LIN {X 0,Y 715.603,Z 787.704,A -85,B 0,C 180,E1 31621.98,E2 31621.98} C_VEL
LIN {X 0,Y 714.708,Z 772.954,A -85,B 0,C 180,E1 31621.864,E2 31621.864} C_VEL
LIN {X 0,Y 714.613,Z 761.128,A -85,B 0,C 180,E1 31621.852,E2 31621.852} C_VEL
LIN {X 0,Y 712.527,Z 773.661,A -85,B 0,C 180,E1 31621.581,E2 31621.581} C_VEL
LIN {X 0,Y 711.718,Z 777.536,A -85,B 0,C 180,E1 31621.475,E2 31621.475} C_VEL
LIN {X 0,Y 707.438,Z 835.712,A -85,B 0,C 180,E1 31620.904,E2 31620.904} C_VEL
LIN {X 0,Y 703.742,Z 875.337,A -85,B 0,C 180,E1 31620.398,E2 31620.398} C_VEL
LIN {X 0,Y 701.35,Z 893.858,A -85,B 0,C 180,E1 31620.063,E2 31620.063} C_VEL
LIN {X 0,Y 699.884,Z 900.884,A -85,B 0,C 180,E1 31619.855,E2 31619.855} C_VEL
LIN {X 0,Y 698.183,Z 921.476,A -85,B 0,C 180,E1 31619.675,E2 31619.675} C_VEL
LIN {X 0,Y 695.199,Z 934.998,A -85,B 0,C 180,E1 31619.546,E2 31619.546} C_VEL
LIN {X 0,Y 691.805,Z 945.388,A -85,B 0,C 180,E1 31619.339,E2 31619.339} C_VEL
LIN {X 0,Y 689.317,Z 952.203,A -85,B 0,C 180,E1 31619.075,E2 31619.075} C_VEL
LIN {X 0,Y 688.817,Z 954.108,A -85,B 0,C 180,E1 31618.988,E2 31618.988} C_VEL
LIN {X 0,Y 688.302,Z 1018.799,A -85,B 0,C 180,E1 31618.229,E2 31618.229} C_VEL
LIN {X 0,Y 687.827,Z 1042.443,A -85,B 0,C 180,E1 31617.796,E2 31617.796} C_VEL
LIN {X 0,Y 687.249,Z 1065.699,A -85,B 0,C 180,E1 31617.208,E2 31617.208} C_VEL
LIN {X 0,Y 686.594,Z 1087.292,A -85,B 0,C 180,E1 31616.511,E2 31616.511} C_VEL
LIN {X 0,Y 685.818,Z 1109.823,A -85,B 0,C 180,E1 31615.613,E2 31615.613} C_VEL
LIN {X 0,Y 685.018,Z 1130.719,A -85,B 0,C 180,E1 31614.616,E2 31614.616} C_VEL
LIN {X 0,Y 684.173,Z 1151.786,A -85,B 0,C 180,E1 31613.424,E2 31613.424} C_VEL
LIN {X 0,Y 683.335,Z 1171.979,A -85,B 0,C 180,E1 31612.09,E2 31612.09} C_VEL
LIN {X 0,Y 682.504,Z 1192.49,A -85,B 0,C 180,E1 31610.497,E2 31610.497} C_VEL
LIN {X 0,Y 681.903,Z 1208.158,A -85,B 0,C 180,E1 31609.087,E2 31609.087} C_VEL
LIN {X 0,Y 681.353,Z 1223.561,A -85,B 0,C 180,E1 31607.509,E2 31607.509} C_VEL
LIN {X 0,Y 680.853,Z 1238.91,A -85,B 0,C 180,E1 31605.678,E2 31605.678} C_VEL
LIN {X 0,Y 680.524,Z 1251.279,A -85,B 0,C 180,E1 31603.944,E2 31603.944} C_VEL
LIN {X 0,Y 680.275,Z 1262.038,A -85,B 0,C 180,E1 31602.192,E2 31602.192} C_VEL
LIN {X 0,Y 680.096,Z 1271.99,A -85,B 0,C 180,E1 31600.248,E2 31600.248} C_VEL
LIN {X 0,Y 679.995,Z 1280.024,A -85,B 0,C 180,E1 31598.286,E2 31598.286} C_VEL
LIN {X 0,Y 679.928,Z 1285.324,A -85,B 0,C 180,E1 31596.673,E2 31596.673} C_VEL
LIN {X 0,Y 679.901,Z 1290.199,A -85,B 0,C 180,E1 31594.725,E2 31594.725} C_VEL
LIN {X 0,Y 679.894,Z 1293.515,A -85,B 0,C 180,E1 31592.614,E2 31592.614} C_VEL
LIN {X 0,Y 679.899,Z 1294.802,A -85,B 0,C 180,E1 31590.76,E2 31590.76} C_VEL
LIN {X 0,Y 679.909,Z 1294.747,A -85,B 0,C 180,E1 31589.074,E2 31589.074} C_VEL
LIN {X 0,Y 679.908,Z 1293.103,A -85,B 0,C 180,E1 31587.051,E2 31587.051} C_VEL
LIN {X 0,Y 679.914,Z 1289.645,A -85,B 0,C 180,E1 31585.024,E2 31585.024} C_VEL
LIN {X 0,Y 679.926,Z 1285.068,A -85,B 0,C 180,E1 31583.245,E2 31583.245} C_VEL
LIN {X 0,Y 679.998,Z 1279.731,A -85,B 0,C 180,E1 31581.631,E2 31581.631} C_VEL
LIN {X 0,Y 680.106,Z 1271.598,A -85,B 0,C 180,E1 31579.669,E2 31579.669} C_VEL
LIN {X 0,Y 680.285,Z 1261.402,A -85,B 0,C 180,E1 31577.696,E2 31577.696} C_VEL
LIN {X 0,Y 680.523,Z 1251.281,A -85,B 0,C 180,E1 31576.058,E2 31576.058} C_VEL
LIN {X 0,Y 680.808,Z 1240.215,A -85,B 0,C 180,E1 31574.498,E2 31574.498} C_VEL
LIN {X 0,Y 681.277,Z 1225.94,A -85,B 0,C 180,E1 31572.756,E2 31572.756} C_VEL
LIN {X 0,Y 681.837,Z 1210.008,A -85,B 0,C 180,E1 31571.091,E2 31571.091} C_VEL
LIN {X 0,Y 682.375,Z 1195.578,A -85,B 0,C 180,E1 31569.77,E2 31569.77} C_VEL
LIN {X 0,Y 683.11,Z 1178.049,A -85,B 0,C 180,E1 31568.353,E2 31568.353} C_VEL
LIN {X 0,Y 683.906,Z 1158.295,A -85,B 0,C 180,E1 31566.979,E2 31566.979} C_VEL
LIN {X 0,Y 684.734,Z 1138.058,A -85,B 0,C 180,E1 31565.776,E2 31565.776} C_VEL
LIN {X 0,Y 685.55,Z 1116.849,A -85,B 0,C 180,E1 31564.702,E2 31564.702} C_VEL
LIN {X 0,Y 686.328,Z 1095.82,A -85,B 0,C 180,E1 31563.806,E2 31563.806} C_VEL
LIN {X 0,Y 687.009,Z 1073.239,A -85,B 0,C 180,E1 31563.019,E2 31563.019} C_VEL
LIN {X 0,Y 687.673,Z 1050.257,A -85,B 0,C 180,E1 31562.385,E2 31562.385} C_VEL
LIN {X 0,Y 688.127,Z 1026.734,A -85,B 0,C 180,E1 31561.899,E2 31561.899} C_VEL
LIN {X 0,Y 688.49,Z 1000.263,A -85,B 0,C 180,E1 31561.535,E2 31561.535} C_VEL
LIN {X 0,Y 688.848,Z 953.484,A -85,B 0,C 180,E1 31561.001,E2 31561.001} C_VEL
LIN {X 0,Y 691.067,Z 947.432,A -85,B 0,C 180,E1 31560.724,E2 31560.724} C_VEL
LIN {X 0,Y 694.4,Z 937.673,A -85,B 0,C 180,E1 31560.494,E2 31560.494} C_VEL
LIN {X 0,Y 697.652,Z 924.638,A -85,B 0,C 180,E1 31560.35,E2 31560.35} C_VEL
LIN {X 0,Y 699.303,Z 910.098,A -85,B 0,C 180,E1 31560.228,E2 31560.228} C_VEL
LIN {X 0,Y 700.088,Z 899.542,A -85,B 0,C 180,E1 31560.116,E2 31560.116} C_VEL
LIN {X 0,Y 701.619,Z 892.218,A -85,B 0,C 180,E1 31559.899,E2 31559.899} C_VEL
LIN {X 0,Y 704.219,Z 870.835,A -85,B 0,C 180,E1 31559.536,E2 31559.536} C_VEL
LIN {X 0,Y 708.05,Z 828.181,A -85,B 0,C 180,E1 31559.013,E2 31559.013} C_VEL
LIN {X 0,Y 711.957,Z 775.957,A -85,B 0,C 180,E1 31558.494,E2 31558.494} C_VEL
LIN {X 0,Y 713.841,Z 766.512,A -85,B 0,C 180,E1 31558.248,E2 31558.248} C_VEL
LIN {X 0,Y 714.629,Z 761.008,A -85,B 0,C 180,E1 31558.146,E2 31558.146} C_VEL
LIN {X 0,Y 714.92,Z 778.455,A -85,B 0,C 180,E1 31558.108,E2 31558.108} C_VEL
LIN {X 0,Y 716.169,Z 792.802,A -85,B 0,C 180,E1 31557.948,E2 31557.948} C_VEL
LIN {X 0,Y 718.366,Z 806.064,A -85,B 0,C 180,E1 31557.669,E2 31557.669} C_VEL
LIN {X 0,Y 721.525,Z 818.398,A -85,B 0,C 180,E1 31557.275,E2 31557.275} C_VEL
LIN {X 0,Y 725.606,Z 829.571,A -85,B 0,C 180,E1 31556.777,E2 31556.777} C_VEL
LIN {X 0,Y 730.214,Z 839.109,A -85,B 0,C 180,E1 31556.203,E2 31556.203} C_VEL
LIN {X 0,Y 731.525,Z 843.469,A -85,B 0,C 180,E1 31555.81,E2 31555.81} C_VEL
LIN {X 0,Y 731.39,Z 846.84,A -85,B 0,C 180,E1 31555.387,E2 31555.387} C_VEL
LIN {X 0,Y 730.13,Z 849.08,A -85,B 0,C 180,E1 31554.979,E2 31554.979} C_VEL
LIN {X 0,Y 727.783,Z 850.434,A -85,B 0,C 180,E1 31554.559,E2 31554.559} C_VEL
LIN {X 0,Y 724.29,Z 850.661,A -85,B 0,C 180,E1 31554.132,E2 31554.132} C_VEL
LIN {X 0,Y 720.235,Z 849.65,A -85,B 0,C 180,E1 31553.765,E2 31553.765} C_VEL
LIN {X 0,Y 711.761,Z 845.351,A -85,B 0,C 180,E1 31553.067,E2 31553.067} C_VEL
LIN {X 0,Y 704.753,Z 839.928,A -85,B 0,C 180,E1 31552.343,E2 31552.343} C_VEL
LIN {X 0,Y 698.647,Z 832.828,A -85,B 0,C 180,E1 31551.523,E2 31551.523} C_VEL
LIN {X 0,Y 694.056,Z 824.409,A -85,B 0,C 180,E1 31550.665,E2 31550.665} C_VEL
LIN {X 0,Y 690.733,Z 814.145,A -85,B 0,C 180,E1 31549.719,E2 31549.719} C_VEL
LIN {X 0,Y 689.006,Z 801.685,A -85,B 0,C 180,E1 31548.68,E2 31548.68} C_VEL
LIN {X 0,Y 688.911,Z 784.149,A -85,B 0,C 180,E1 31547.33,E2 31547.33} C_VEL
LIN {X 0,Y 690.246,Z 746.13,A -85,B 0,C 180,E1 31544.428,E2 31544.428} C_VEL
LIN {X 0,Y 691.594,Z 709.846,A -85,B 0,C 180,E1 31541.576,E2 31541.576} C_VEL
LIN {X 0,Y 692.854,Z 674.643,A -85,B 0,C 180,E1 31538.727,E2 31538.727} C_VEL
LIN {X 0,Y 694.016,Z 640.169,A -85,B 0,C 180,E1 31535.845,E2 31535.845} C_VEL
LIN {X 0,Y 694.079,Z 634.852,A -85,B 0,C 180,E1 31535.378,E2 31535.378} C_VEL
LIN {X 0,Y 685.307,Z 614.541,A -85,B 0,C 180,E1 31532.773,E2 31532.773} C_VEL
LIN {X 0,Y 681.315,Z 605.83,A -85,B 0,C 180,E1 31531.596,E2 31531.596} C_VEL
LIN {X 0,Y 680.505,Z 603.217,A -85,B 0,C 180,E1 31531.244,E2 31531.244} C_VEL
LIN {X 0,Y 680.512,Z 603.214,A -85,B 0,C 180,E1 31528.333,E2 31528.333} C_VEL
LIN {X 0,Y 680.516,Z 603.213,A -85,B 0,C 180,E1 31525.314,E2 31525.314} C_VEL
LIN {X 0,Y 680.519,Z 603.213,A -85,B 0,C 180,E1 31522.237,E2 31522.237} C_VEL
LIN {X 0,Y 680.52,Z 603.21,A -85,B 0,C 180,E1 31519.127,E2 31519.127} C_VEL
LIN {X 0,Y 680.521,Z 603.213,A -85,B 0,C 180,E1 31516.035,E2 31516.035} C_VEL
LIN {X 0,Y 680.524,Z 603.212,A -85,B 0,C 180,E1 31512.991,E2 31512.991} C_VEL
LIN {X 0,Y 680.526,Z 603.215,A -85,B 0,C 180,E1 31509.899,E2 31509.899} C_VEL
LIN {X 0,Y 680.53,Z 603.213,A -85,B 0,C 180,E1 31506.835,E2 31506.835} C_VEL
LIN {X 0,Y 680.515,Z 603.214,A -85,B 0,C 180,E1 31503.791,E2 31503.791} C_VEL
LIN {X 0,Y 680.511,Z 603.212,A -85,B 0,C 180,E1 31500.758,E2 31500.758} C_VEL
LIN {X 0,Y 680.505,Z 603.211,A -85,B 0,C 180,E1 31497.811,E2 31497.811} C_VEL
LIN {X 0,Y 680.504,Z 603.211,A -85,B 0,C 180,E1 31494.858,E2 31494.858} C_VEL
LIN {X 0,Y 680.508,Z 603.211,A -85,B 0,C 180,E1 31491.891,E2 31491.891} C_VEL
LIN {X 0,Y 680.515,Z 603.211,A -85,B 0,C 180,E1 31488.902,E2 31488.902} C_VEL
LIN {X 0,Y 680.522,Z 603.212,A -85,B 0,C 180,E1 31485.86,E2 31485.86} C_VEL
LIN {X 0,Y 680.521,Z 603.213,A -85,B 0,C 180,E1 31482.734,E2 31482.734} C_VEL
LIN {X 0,Y 680.524,Z 603.213,A -85,B 0,C 180,E1 31479.711,E2 31479.711} C_VEL
LIN {X 0,Y 680.526,Z 603.212,A -85,B 0,C 180,E1 31476.627,E2 31476.627} C_VEL
LIN {X 0,Y 680.522,Z 603.215,A -85,B 0,C 180,E1 31473.564,E2 31473.564} C_VEL
LIN {X 0,Y 680.511,Z 603.214,A -85,B 0,C 180,E1 31470.607,E2 31470.607} C_VEL
LIN {X 0,Y 680.52,Z 603.208,A -85,B 0,C 180,E1 31469.429,E2 31469.429} C_VEL
LIN {X 0,Y 679.55,Z 603.333,A -85,B 0,C 180,E1 31468.78,E2 31468.78} C_VEL
LIN {X 0,Y 673.093,Z 604.139,A -85,B 0,C 180,E1 31466.963,E2 31466.963} C_VEL
LIN {X 0,Y 672.574,Z 604.199,A -85,B 0,C 180,E1 31466.49,E2 31466.49} C_VEL
LIN {X 0,Y 672.566,Z 604.202,A -85,B 0,C 180,E1 31463.511,E2 31463.511} C_VEL
LIN {X 0,Y 672.583,Z 604.204,A -85,B 0,C 180,E1 31460.595,E2 31460.595} C_VEL
LIN {X 0,Y 672.576,Z 604.194,A -85,B 0,C 180,E1 31457.55,E2 31457.55} C_VEL
LIN {X 0,Y 672.586,Z 604.2,A -85,B 0,C 180,E1 31454.56,E2 31454.56} C_VEL
LIN {X 0,Y 672.591,Z 604.193,A -85,B 0,C 180,E1 31451.416,E2 31451.416} C_VEL
LIN {X 0,Y 672.579,Z 604.203,A -85,B 0,C 180,E1 31448.283,E2 31448.283} C_VEL
LIN {X 0,Y 672.591,Z 604.204,A -85,B 0,C 180,E1 31445.15,E2 31445.15} C_VEL
LIN {X 0,Y 672.576,Z 604.205,A -85,B 0,C 180,E1 31442.053,E2 31442.053} C_VEL
LIN {X 0,Y 672.594,Z 604.397,A -85,B 0,C 180,E1 31440.786,E2 31440.786} C_VEL
LIN {X 0,Y 677.704,Z 621.502,A -85,B 0,C 180,E1 31439.484,E2 31439.484} C_VEL
LIN {X 0,Y 677.378,Z 660.167,A -85,B 0,C 180,E1 31436.945,E2 31436.945} C_VEL
LIN {X 0,Y 676.584,Z 704.691,A -85,B 0,C 180,E1 31433.978,E2 31433.978} C_VEL
LIN {X 0,Y 675.775,Z 749.981,A -85,B 0,C 180,E1 31430.98,E2 31430.98} C_VEL
LIN {X 0,Y 674.803,Z 795.336,A -85,B 0,C 180,E1 31427.95,E2 31427.95} C_VEL
LIN {X 0,Y 674.169,Z 831.281,A -85,B 0,C 180,E1 31425.589,E2 31425.589} C_VEL
LIN {X 0,Y 675.101,Z 841.648,A -85,B 0,C 180,E1 31425.451,E2 31425.451} C_VEL
LIN {X 0,Y 674.416,Z 1000.774,A -85,B 0,C 180,E1 31423.715,E2 31423.715} C_VEL
LIN {X 0,Y 674.227,Z 1018.235,A -85,B 0,C 180,E1 31423.37,E2 31423.37} C_VEL
LIN {X 0,Y 673.939,Z 1035.447,A -85,B 0,C 180,E1 31422.857,E2 31422.857} C_VEL
LIN {X 0,Y 673.617,Z 1051.632,A -85,B 0,C 180,E1 31422.21,E2 31422.21} C_VEL
LIN {X 0,Y 673.284,Z 1066.92,A -85,B 0,C 180,E1 31421.43,E2 31421.43} C_VEL
LIN {X 0,Y 672.954,Z 1081.016,A -85,B 0,C 180,E1 31420.529,E2 31420.529} C_VEL
LIN {X 0,Y 672.636,Z 1094.67,A -85,B 0,C 180,E1 31419.453,E2 31419.453} C_VEL
LIN {X 0,Y 672.382,Z 1106.683,A -85,B 0,C 180,E1 31418.292,E2 31418.292} C_VEL
LIN {X 0,Y 672.193,Z 1116.775,A -85,B 0,C 180,E1 31417.091,E2 31417.091} C_VEL
LIN {X 0,Y 672.051,Z 1125.967,A -85,B 0,C 180,E1 31415.72,E2 31415.72} C_VEL
LIN {X 0,Y 671.974,Z 1133.125,A -85,B 0,C 180,E1 31414.351,E2 31414.351} C_VEL
LIN {X 0,Y 671.934,Z 1138.766,A -85,B 0,C 180,E1 31412.899,E2 31412.899} C_VEL
LIN {X 0,Y 671.917,Z 1142.505,A -85,B 0,C 180,E1 31411.448,E2 31411.448} C_VEL
LIN {X 0,Y 671.924,Z 1144.6,A -85,B 0,C 180,E1 31409.914,E2 31409.914} C_VEL
LIN {X 0,Y 671.914,Z 1144.855,A -85,B 0,C 180,E1 31408.379,E2 31408.379} C_VEL
LIN {X 0,Y 671.919,Z 1143.303,A -85,B 0,C 180,E1 31406.892,E2 31406.892} C_VEL
LIN {X 0,Y 671.925,Z 1139.885,A -85,B 0,C 180,E1 31405.39,E2 31405.39} C_VEL
LIN {X 0,Y 671.96,Z 1134.758,A -85,B 0,C 180,E1 31403.934,E2 31403.934} C_VEL
LIN {X 0,Y 672.026,Z 1128.128,A -85,B 0,C 180,E1 31402.561,E2 31402.561} C_VEL
LIN {X 0,Y 672.14,Z 1120.07,A -85,B 0,C 180,E1 31401.271,E2 31401.271} C_VEL
LIN {X 0,Y 672.316,Z 1109.903,A -85,B 0,C 180,E1 31399.978,E2 31399.978} C_VEL
LIN {X 0,Y 672.56,Z 1098.153,A -85,B 0,C 180,E1 31398.768,E2 31398.768} C_VEL
LIN {X 0,Y 672.86,Z 1085.21,A -85,B 0,C 180,E1 31397.686,E2 31397.686} C_VEL
LIN {X 0,Y 673.185,Z 1071.123,A -85,B 0,C 180,E1 31396.733,E2 31396.733} C_VEL
LIN {X 0,Y 673.522,Z 1056.055,A -85,B 0,C 180,E1 31395.908,E2 31395.908} C_VEL
LIN {X 0,Y 673.857,Z 1039.951,A -85,B 0,C 180,E1 31395.212,E2 31395.212} C_VEL
LIN {X 0,Y 674.151,Z 1022.973,A -85,B 0,C 180,E1 31394.666,E2 31394.666} C_VEL
LIN {X 0,Y 674.374,Z 1004.976,A -85,B 0,C 180,E1 31394.264,E2 31394.264} C_VEL
LIN {X 0,Y 674.515,Z 984.639,A -85,B 0,C 180,E1 31393.999,E2 31393.999} C_VEL
LIN {X 0,Y 674.892,Z 837.233,A -85,B 0,C 180,E1 31392.406,E2 31392.406} C_VEL
LIN {X 0,Y 674.157,Z 830.801,A -85,B 0,C 180,E1 31392.298,E2 31392.298} C_VEL
LIN {X 0,Y 675.054,Z 785.156,A -85,B 0,C 180,E1 31389.267,E2 31389.267} C_VEL
LIN {X 0,Y 675.759,Z 751.14,A -85,B 0,C 180,E1 31387.005,E2 31387.005} C_VEL
LIN {X 0,Y 676.57,Z 705.123,A -85,B 0,C 180,E1 31383.963,E2 31383.963} C_VEL
LIN {X 0,Y 677.378,Z 659.877,A -85,B 0,C 180,E1 31380.945,E2 31380.945} C_VEL
LIN {X 0,Y 677.729,Z 621.412,A -85,B 0,C 180,E1 31378.415,E2 31378.415} C_VEL
LIN {X 0,Y 672.578,Z 604.201,A -85,B 0,C 180,E1 31377.086,E2 31377.086} C_VEL
LIN {X 0,Y 672.567,Z 604.197,A -85,B 0,C 180,E1 31374.038,E2 31374.038} C_VEL
LIN {X 0,Y 672.588,Z 604.195,A -85,B 0,C 180,E1 31371.033,E2 31371.033} C_VEL
LIN {X 0,Y 672.567,Z 604.198,A -85,B 0,C 180,E1 31368.009,E2 31368.009} C_VEL
LIN {X 0,Y 672.576,Z 604.202,A -85,B 0,C 180,E1 31365.044,E2 31365.044} C_VEL
LIN {X 0,Y 672.584,Z 604.196,A -85,B 0,C 180,E1 31361.984,E2 31361.984} C_VEL
LIN {X 0,Y 672.579,Z 604.2,A -85,B 0,C 180,E1 31358.856,E2 31358.856} C_VEL
LIN {X 0,Y 672.589,Z 604.203,A -85,B 0,C 180,E1 31355.75,E2 31355.75} C_VEL
LIN {X 0,Y 672.583,Z 604.204,A -85,B 0,C 180,E1 31352.66,E2 31352.66} C_VEL
LIN {X 0,Y 672.579,Z 604.3,A -85,B 0,C 180,E1 31350.233,E2 31350.233} C_VEL
LIN {X 0,Y 672.874,Z 605.616,A -85,B 0,C 180,E1 31350.149,E2 31350.149} C_VEL
LIN {X 0,Y 674.8,Z 608.814,A -85,B 0,C 180,E1 31349.992,E2 31349.992} C_VEL
LIN {X 0,Y 683.922,Z 625.294,A -85,B 0,C 180,E1 31349.274,E2 31349.274} C_VEL
LIN {X 0,Y 681.83,Z 883.098,A -85,B 0,C 180,E1 31346.28,E2 31346.28} C_VEL
LIN {X 0,Y 681.257,Z 946.678,A -85,B 0,C 180,E1 31345.528,E2 31345.528} C_VEL
LIN {X 0,Y 680.809,Z 970.073,A -85,B 0,C 180,E1 31345.119,E2 31345.119} C_VEL
LIN {X 0,Y 680.146,Z 992.867,A -85,B 0,C 180,E1 31344.552,E2 31344.552} C_VEL
LIN {X 0,Y 679.55,Z 1011.718,A -85,B 0,C 180,E1 31343.961,E2 31343.961} C_VEL
LIN {X 0,Y 678.871,Z 1029.536,A -85,B 0,C 180,E1 31343.295,E2 31343.295} C_VEL
LIN {X 0,Y 678.195,Z 1046.859,A -85,B 0,C 180,E1 31342.54,E2 31342.54} C_VEL
LIN {X 0,Y 677.316,Z 1067.83,A -85,B 0,C 180,E1 31341.476,E2 31341.476} C_VEL
LIN {X 0,Y 676.37,Z 1088.323,A -85,B 0,C 180,E1 31340.239,E2 31340.239} C_VEL
LIN {X 0,Y 675.609,Z 1104.819,A -85,B 0,C 180,E1 31339.092,E2 31339.092} C_VEL
LIN {X 0,Y 674.944,Z 1119.984,A -85,B 0,C 180,E1 31337.903,E2 31337.903} C_VEL
LIN {X 0,Y 674.231,Z 1136.28,A -85,B 0,C 180,E1 31336.455,E2 31336.455} C_VEL
LIN {X 0,Y 673.511,Z 1154.036,A -85,B 0,C 180,E1 31334.619,E2 31334.619} C_VEL
LIN {X 0,Y 673.049,Z 1167.097,A -85,B 0,C 180,E1 31333.051,E2 31333.051} C_VEL
LIN {X 0,Y 672.652,Z 1179.65,A -85,B 0,C 180,E1 31331.316,E2 31331.316} C_VEL
LIN {X 0,Y 672.338,Z 1191.404,A -85,B 0,C 180,E1 31329.415,E2 31329.415} C_VEL
LIN {X 0,Y 672.128,Z 1201.454,A -85,B 0,C 180,E1 31327.436,E2 31327.436} C_VEL
LIN {X 0,Y 672.003,Z 1209.282,A -85,B 0,C 180,E1 31325.55,E2 31325.55} C_VEL
LIN {X 0,Y 671.948,Z 1215.203,A -85,B 0,C 180,E1 31323.754,E2 31323.754} C_VEL
LIN {X 0,Y 671.916,Z 1220.399,A -85,B 0,C 180,E1 31321.62,E2 31321.62} C_VEL
LIN {X 0,Y 671.904,Z 1223.334,A -85,B 0,C 180,E1 31319.744,E2 31319.744} C_VEL
LIN {X 0,Y 671.904,Z 1224.787,A -85,B 0,C 180,E1 31317.783,E2 31317.783} C_VEL
LIN {X 0,Y 671.912,Z 1224.731,A -85,B 0,C 180,E1 31315.989,E2 31315.989} C_VEL
LIN {X 0,Y 671.919,Z 1223.059,A -85,B 0,C 180,E1 31313.935,E2 31313.935} C_VEL
LIN {X 0,Y 671.928,Z 1219.534,A -85,B 0,C 180,E1 31311.873,E2 31311.873} C_VEL
LIN {X 0,Y 671.955,Z 1214.979,A -85,B 0,C 180,E1 31310.091,E2 31310.091} C_VEL
LIN {X 0,Y 672.005,Z 1209.462,A -85,B 0,C 180,E1 31308.412,E2 31308.412} C_VEL
LIN {X 0,Y 672.128,Z 1201.571,A -85,B 0,C 180,E1 31306.493,E2 31306.493} C_VEL
LIN {X 0,Y 672.337,Z 1191.242,A -85,B 0,C 180,E1 31304.473,E2 31304.473} C_VEL
LIN {X 0,Y 672.608,Z 1180.95,A -85,B 0,C 180,E1 31302.793,E2 31302.793} C_VEL
LIN {X 0,Y 672.957,Z 1169.634,A -85,B 0,C 180,E1 31301.19,E2 31301.19} C_VEL
LIN {X 0,Y 673.434,Z 1156.207,A -85,B 0,C 180,E1 31299.536,E2 31299.536} C_VEL
LIN {X 0,Y 674.137,Z 1138.647,A -85,B 0,C 180,E1 31297.685,E2 31297.685} C_VEL
LIN {X 0,Y 674.778,Z 1123.633,A -85,B 0,C 180,E1 31296.314,E2 31296.314} C_VEL
LIN {X 0,Y 675.517,Z 1107.29,A -85,B 0,C 180,E1 31295.001,E2 31295.001} C_VEL
LIN {X 0,Y 676.327,Z 1089.423,A -85,B 0,C 180,E1 31293.741,E2 31293.741} C_VEL
LIN {X 0,Y 677.304,Z 1067.704,A -85,B 0,C 180,E1 31292.431,E2 31292.431} C_VEL
LIN {X 0,Y 678.102,Z 1048.803,A -85,B 0,C 180,E1 31291.461,E2 31291.461} C_VEL
LIN {X 0,Y 678.798,Z 1031.547,A -85,B 0,C 180,E1 31290.697,E2 31290.697} C_VEL
LIN {X 0,Y 679.463,Z 1013.908,A -85,B 0,C 180,E1 31290.026,E2 31290.026} C_VEL
LIN {X 0,Y 680.056,Z 995.914,A -85,B 0,C 180,E1 31289.448,E2 31289.448} C_VEL
LIN {X 0,Y 680.649,Z 975.131,A -85,B 0,C 180,E1 31288.906,E2 31288.906} C_VEL
LIN {X 0,Y 681.229,Z 949.547,A -85,B 0,C 180,E1 31288.422,E2 31288.422} C_VEL
LIN {X 0,Y 681.625,Z 909.928,A -85,B 0,C 180,E1 31287.937,E2 31287.937} C_VEL
LIN {X 0,Y 683.667,Z 645.309,A -85,B 0,C 180,E1 31284.885,E2 31284.885} C_VEL
LIN {X 0,Y 683.579,Z 624.804,A -85,B 0,C 180,E1 31284.653,E2 31284.653} C_VEL
LIN {X 0,Y 675.913,Z 612.154,A -85,B 0,C 180,E1 31284.244,E2 31284.244} C_VEL
LIN {X 0,Y 675.178,Z 610.975,A -85,B 0,C 180,E1 31283.386,E2 31283.386} C_VEL
LIN {X 0,Y 675.379,Z 611.387,A -85,B 0,C 180,E1 31282.199,E2 31282.199} C_VEL
LIN {X 0,Y 676.034,Z 612.93,A -85,B 0,C 180,E1 31281.271,E2 31281.271} C_VEL
LIN {X 0,Y 677.44,Z 616.483,A -85,B 0,C 180,E1 31280.055,E2 31280.055} C_VEL
LIN {X 0,Y 678.902,Z 620.462,A -85,B 0,C 180,E1 31279.161,E2 31279.161} C_VEL
LIN {X 0,Y 679.568,Z 622.879,A -85,B 0,C 180,E1 31278.753,E2 31278.753} C_VEL
LIN {X 0,Y 676.672,Z 634.327,A -85,B 0,C 180,E1 31277.752,E2 31277.752} C_VEL
LIN {X 0,Y 674.724,Z 648.114,A -85,B 0,C 180,E1 31276.756,E2 31276.756} C_VEL
LIN {X 0,Y 673.436,Z 666.247,A -85,B 0,C 180,E1 31275.66,E2 31275.66} C_VEL
LIN {X 0,Y 672.583,Z 694.895,A -85,B 0,C 180,E1 31274.161,E2 31274.161} C_VEL
LIN {X 0,Y 672.595,Z 770.126,A -85,B 0,C 180,E1 31270.516,E2 31270.516} C_VEL
LIN {X 0,Y 674.512,Z 789.281,A -85,B 0,C 180,E1 31269.57,E2 31269.57} C_VEL
LIN {X 0,Y 677.902,Z 804.887,A -85,B 0,C 180,E1 31268.782,E2 31268.782} C_VEL
LIN {X 0,Y 682.915,Z 818.369,A -85,B 0,C 180,E1 31268.095,E2 31268.095} C_VEL
LIN {X 0,Y 689.341,Z 830.207,A -85,B 0,C 180,E1 31267.493,E2 31267.493} C_VEL
LIN {X 0,Y 697.093,Z 840.45,A -85,B 0,C 180,E1 31266.97,E2 31266.97} C_VEL
LIN {X 0,Y 705.641,Z 848.966,A -85,B 0,C 180,E1 31266.54,E2 31266.54} C_VEL
LIN {X 0,Y 710.972,Z 853.164,A -85,B 0,C 180,E1 31266.307,E2 31266.307} C_VEL
LIN {X 0,Y 715.788,Z 855.733,A -85,B 0,C 180,E1 31266.02,E2 31266.02} C_VEL
LIN {X 0,Y 720.755,Z 857.13,A -85,B 0,C 180,E1 31265.615,E2 31265.615} C_VEL
LIN {X 0,Y 724.417,Z 857.036,A -85,B 0,C 180,E1 31265.202,E2 31265.202} C_VEL
LIN {X 0,Y 726.939,Z 855.868,A -85,B 0,C 180,E1 31264.798,E2 31264.798} C_VEL
LIN {X 0,Y 728.59,Z 853.457,A -85,B 0,C 180,E1 31264.336,E2 31264.336} C_VEL
LIN {X 0,Y 728.825,Z 849.868,A -85,B 0,C 180,E1 31263.877,E2 31263.877} C_VEL
LIN {X 0,Y 727.476,Z 845.421,A -85,B 0,C 180,E1 31263.471,E2 31263.471} C_VEL
LIN {X 0,Y 722.555,Z 835.393,A -85,B 0,C 180,E1 31262.852,E2 31262.852} C_VEL
LIN {X 0,Y 718.281,Z 823.93,A -85,B 0,C 180,E1 31262.32,E2 31262.32} C_VEL
LIN {X 0,Y 714.893,Z 811.222,A -85,B 0,C 180,E1 31261.888,E2 31261.888} C_VEL
LIN {X 0,Y 713.904,Z 806.816,A -85,B 0,C 180,E1 31261.761,E2 31261.761} C_VEL
LIN {X 0,Y 709.694,Z 857.632,A -85,B 0,C 180,E1 31261.207,E2 31261.207} C_VEL
LIN {X 0,Y 706.453,Z 887.77,A -85,B 0,C 180,E1 31260.77,E2 31260.77} C_VEL
LIN {X 0,Y 704.454,Z 900.073,A -85,B 0,C 180,E1 31260.499,E2 31260.499} C_VEL
LIN {X 0,Y 703.692,Z 903.617,A -85,B 0,C 180,E1 31260.403,E2 31260.403} C_VEL
LIN {X 0,Y 701.396,Z 917.517,A -85,B 0,C 180,E1 31260.329,E2 31260.329} C_VEL
LIN {X 0,Y 697.161,Z 931.222,A -85,B 0,C 180,E1 31260.251,E2 31260.251} C_VEL
LIN {X 0,Y 692.222,Z 942.907,A -85,B 0,C 180,E1 31260.082,E2 31260.082} C_VEL
LIN {X 0,Y 688.44,Z 951.342,A -85,B 0,C 180,E1 31259.832,E2 31259.832} C_VEL
LIN {X 0,Y 686.29,Z 956.568,A -85,B 0,C 180,E1 31259.598,E2 31259.598} C_VEL
LIN {X 0,Y 683.145,Z 963.389,A -85,B 0,C 180,E1 31259.363,E2 31259.363} C_VEL
LIN {X 0,Y 681.716,Z 967.596,A -85,B 0,C 180,E1 31259.159,E2 31259.159} C_VEL
LIN {X 0,Y 681.239,Z 1019.137,A -85,B 0,C 180,E1 31258.543,E2 31258.543} C_VEL
LIN {X 0,Y 680.727,Z 1042.437,A -85,B 0,C 180,E1 31258.112,E2 31258.112} C_VEL
LIN {X 0,Y 680.09,Z 1065.619,A -85,B 0,C 180,E1 31257.521,E2 31257.521} C_VEL
LIN {X 0,Y 679.369,Z 1087.285,A -85,B 0,C 180,E1 31256.815,E2 31256.815} C_VEL
LIN {X 0,Y 678.499,Z 1109.822,A -85,B 0,C 180,E1 31255.91,E2 31255.91} C_VEL
LIN {X 0,Y 677.595,Z 1131.325,A -85,B 0,C 180,E1 31254.871,E2 31254.871} C_VEL
LIN {X 0,Y 676.649,Z 1152.515,A -85,B 0,C 180,E1 31253.654,E2 31253.654} C_VEL
LIN {X 0,Y 675.726,Z 1172.599,A -85,B 0,C 180,E1 31252.307,E2 31252.307} C_VEL
LIN {X 0,Y 674.832,Z 1192.485,A -85,B 0,C 180,E1 31250.741,E2 31250.741} C_VEL
LIN {X 0,Y 674.187,Z 1207.348,A -85,B 0,C 180,E1 31249.394,E2 31249.394} C_VEL
LIN {X 0,Y 673.599,Z 1221.925,A -85,B 0,C 180,E1 31247.896,E2 31247.896} C_VEL
LIN {X 0,Y 673.108,Z 1235.464,A -85,B 0,C 180,E1 31246.306,E2 31246.306} C_VEL
LIN {X 0,Y 672.648,Z 1249.555,A -85,B 0,C 180,E1 31244.375,E2 31244.375} C_VEL
LIN {X 0,Y 672.365,Z 1260.005,A -85,B 0,C 180,E1 31242.694,E2 31242.694} C_VEL
LIN {X 0,Y 672.153,Z 1269.959,A -85,B 0,C 180,E1 31240.804,E2 31240.804} C_VEL
LIN {X 0,Y 672.006,Z 1278.797,A -85,B 0,C 180,E1 31238.73,E2 31238.73} C_VEL
LIN {X 0,Y 671.937,Z 1284.826,A -85,B 0,C 180,E1 31236.924,E2 31236.924} C_VEL
LIN {X 0,Y 671.924,Z 1289.439,A -85,B 0,C 180,E1 31235.124,E2 31235.124} C_VEL
LIN {X 0,Y 671.911,Z 1292.878,A -85,B 0,C 180,E1 31233.157,E2 31233.157} C_VEL
LIN {X 0,Y 671.909,Z 1294.692,A -85,B 0,C 180,E1 31231.11,E2 31231.11} C_VEL
LIN {X 0,Y 671.895,Z 1294.826,A -85,B 0,C 180,E1 31229.319,E2 31229.319} C_VEL
LIN {X 0,Y 671.894,Z 1293.586,A -85,B 0,C 180,E1 31227.442,E2 31227.442} C_VEL
LIN {X 0,Y 671.901,Z 1290.679,A -85,B 0,C 180,E1 31225.478,E2 31225.478} C_VEL
LIN {X 0,Y 671.93,Z 1285.822,A -85,B 0,C 180,E1 31223.422,E2 31223.422} C_VEL
LIN {X 0,Y 672.002,Z 1280.269,A -85,B 0,C 180,E1 31221.681,E2 31221.681} C_VEL
LIN {X 0,Y 672.104,Z 1272.765,A -85,B 0,C 180,E1 31219.804,E2 31219.804} C_VEL
LIN {X 0,Y 672.317,Z 1262.403,A -85,B 0,C 180,E1 31217.722,E2 31217.722} C_VEL
LIN {X 0,Y 672.587,Z 1251.852,A -85,B 0,C 180,E1 31215.978,E2 31215.978} C_VEL
LIN {X 0,Y 672.884,Z 1241.509,A -85,B 0,C 180,E1 31214.487,E2 31214.487} C_VEL
LIN {X 0,Y 673.369,Z 1228.24,A -85,B 0,C 180,E1 31212.814,E2 31212.814} C_VEL
LIN {X 0,Y 674.01,Z 1211.831,A -85,B 0,C 180,E1 31211.043,E2 31211.043} C_VEL
LIN {X 0,Y 674.636,Z 1196.593,A -85,B 0,C 180,E1 31209.618,E2 31209.618} C_VEL
LIN {X 0,Y 675.351,Z 1180.927,A -85,B 0,C 180,E1 31208.323,E2 31208.323} C_VEL
LIN {X 0,Y 676.168,Z 1162.989,A -85,B 0,C 180,E1 31207.023,E2 31207.023} C_VEL
LIN {X 0,Y 677.128,Z 1142.029,A -85,B 0,C 180,E1 31205.718,E2 31205.718} C_VEL
LIN {X 0,Y 678.004,Z 1121.62,A -85,B 0,C 180,E1 31204.637,E2 31204.637} C_VEL
LIN {X 0,Y 678.885,Z 1100.316,A -85,B 0,C 180,E1 31203.685,E2 31203.685} C_VEL
LIN {X 0,Y 679.703,Z 1077.538,A -85,B 0,C 180,E1 31202.846,E2 31202.846} C_VEL
LIN {X 0,Y 680.442,Z 1054.302,A -85,B 0,C 180,E1 31202.169,E2 31202.169} C_VEL
LIN {X 0,Y 681.009,Z 1030.794,A -85,B 0,C 180,E1 31201.653,E2 31201.653} C_VEL
LIN {X 0,Y 681.407,Z 1006.439,A -85,B 0,C 180,E1 31201.285,E2 31201.285} C_VEL
LIN {X 0,Y 681.816,Z 966.846,A -85,B 0,C 180,E1 31200.818,E2 31200.818} C_VEL
LIN {X 0,Y 684.517,Z 960.279,A -85,B 0,C 180,E1 31200.512,E2 31200.512} C_VEL
LIN {X 0,Y 686.897,Z 955.104,A -85,B 0,C 180,E1 31200.337,E2 31200.337} C_VEL
LIN {X 0,Y 690.231,Z 947.297,A -85,B 0,C 180,E1 31200.03,E2 31200.03} C_VEL
LIN {X 0,Y 694.971,Z 936.664,A -85,B 0,C 180,E1 31199.809,E2 31199.809} C_VEL
LIN {X 0,Y 699.758,Z 923.61,A -85,B 0,C 180,E1 31199.699,E2 31199.699} C_VEL
LIN {X 0,Y 702.914,Z 909.76,A -85,B 0,C 180,E1 31199.635,E2 31199.635} C_VEL
LIN {X 0,Y 703.946,Z 902.104,A -85,B 0,C 180,E1 31199.567,E2 31199.567} C_VEL
LIN {X 0,Y 705.792,Z 892.558,A -85,B 0,C 180,E1 31199.32,E2 31199.32} C_VEL
LIN {X 0,Y 708.614,Z 868.663,A -85,B 0,C 180,E1 31198.937,E2 31198.937} C_VEL
LIN {X 0,Y 712.602,Z 823.803,A -85,B 0,C 180,E1 31198.409,E2 31198.409} C_VEL
LIN {X 0,Y 713.956,Z 806.694,A -85,B 0,C 180,E1 31198.233,E2 31198.233} C_VEL
LIN {X 0,Y 716.999,Z 819.641,A -85,B 0,C 180,E1 31197.842,E2 31197.842} C_VEL
LIN {X 0,Y 720.985,Z 831.587,A -85,B 0,C 180,E1 31197.342,E2 31197.342} C_VEL
LIN {X 0,Y 725.812,Z 842.181,A -85,B 0,C 180,E1 31196.752,E2 31196.752} C_VEL
LIN {X 0,Y 728.187,Z 847.231,A -85,B 0,C 180,E1 31196.38,E2 31196.38} C_VEL
LIN {X 0,Y 728.92,Z 851.382,A -85,B 0,C 180,E1 31195.949,E2 31195.949} C_VEL
LIN {X 0,Y 728.103,Z 854.535,A -85,B 0,C 180,E1 31195.485,E2 31195.485} C_VEL
LIN {X 0,Y 726.001,Z 856.473,A -85,B 0,C 180,E1 31195.032,E2 31195.032} C_VEL
LIN {X 0,Y 722.662,Z 857.237,A -85,B 0,C 180,E1 31194.583,E2 31194.583} C_VEL
LIN {X 0,Y 718.712,Z 856.729,A -85,B 0,C 180,E1 31194.202,E2 31194.202} C_VEL
LIN {X 0,Y 710,Z 853.096,A -85,B 0,C 180,E1 31193.527,E2 31193.527} C_VEL
LIN {X 0,Y 701.281,Z 847.36,A -85,B 0,C 180,E1 31192.704,E2 31192.704} C_VEL
LIN {X 0,Y 694.253,Z 840.304,A -85,B 0,C 180,E1 31191.842,E2 31191.842} C_VEL
LIN {X 0,Y 688.855,Z 831.985,A -85,B 0,C 180,E1 31190.948,E2 31190.948} C_VEL
LIN {X 0,Y 684.68,Z 821.421,A -85,B 0,C 180,E1 31189.928,E2 31189.928} C_VEL
LIN {X 0,Y 682.325,Z 809.279,A -85,B 0,C 180,E1 31188.871,E2 31188.871} C_VEL
LIN {X 0,Y 681.652,Z 792.916,A -85,B 0,C 180,E1 31187.567,E2 31187.567} C_VEL
LIN {X 0,Y 683.186,Z 752.785,A -85,B 0,C 180,E1 31184.489,E2 31184.489} C_VEL
LIN {X 0,Y 684.647,Z 716.285,A -85,B 0,C 180,E1 31181.607,E2 31181.607} C_VEL
LIN {X 0,Y 686.025,Z 681.319,A -85,B 0,C 180,E1 31178.763,E2 31178.763} C_VEL
LIN {X 0,Y 687.364,Z 646.478,A -85,B 0,C 180,E1 31175.839,E2 31175.839} C_VEL
LIN {X 0,Y 687.465,Z 638.789,A -85,B 0,C 180,E1 31175.168,E2 31175.168} C_VEL
LIN {X 0,Y 678.881,Z 619,A -85,B 0,C 180,E1 31172.602,E2 31172.602} C_VEL
LIN {X 0,Y 673.634,Z 607.307,A -85,B 0,C 180,E1 31171.002,E2 31171.002} C_VEL
LIN {X 0,Y 672.581,Z 604.2,A -85,B 0,C 180,E1 31170.56,E2 31170.56} C_VEL
LIN {X 0,Y 672.586,Z 604.201,A -85,B 0,C 180,E1 31167.539,E2 31167.539} C_VEL
LIN {X 0,Y 672.586,Z 604.202,A -85,B 0,C 180,E1 31164.505,E2 31164.505} C_VEL
LIN {X 0,Y 672.586,Z 604.204,A -85,B 0,C 180,E1 31161.36,E2 31161.36} C_VEL
LIN {X 0,Y 672.583,Z 604.201,A -85,B 0,C 180,E1 31158.281,E2 31158.281} C_VEL
LIN {X 0,Y 672.583,Z 604.202,A -85,B 0,C 180,E1 31155.168,E2 31155.168} C_VEL
LIN {X 0,Y 672.585,Z 604.2,A -85,B 0,C 180,E1 31152.013,E2 31152.013} C_VEL
LIN {X 0,Y 672.583,Z 604.201,A -85,B 0,C 180,E1 31148.808,E2 31148.808} C_VEL
LIN {X 0,Y 672.589,Z 604.197,A -85,B 0,C 180,E1 31145.631,E2 31145.631} C_VEL
LIN {X 0,Y 672.578,Z 604.201,A -85,B 0,C 180,E1 31142.471,E2 31142.471} C_VEL
LIN {X 0,Y 672.588,Z 604.2,A -85,B 0,C 180,E1 31139.319,E2 31139.319} C_VEL
LIN {X 0,Y 672.576,Z 604.201,A -85,B 0,C 180,E1 31136.164,E2 31136.164} C_VEL
LIN {X 0,Y 672.588,Z 604.198,A -85,B 0,C 180,E1 31133.084,E2 31133.084} C_VEL
LIN {X 0,Y 672.58,Z 604.198,A -85,B 0,C 180,E1 31129.983,E2 31129.983} C_VEL
LIN {X 0,Y 672.584,Z 604.197,A -85,B 0,C 180,E1 31126.834,E2 31126.834} C_VEL
LIN {X 0,Y 672.58,Z 604.197,A -85,B 0,C 180,E1 31123.77,E2 31123.77} C_VEL
LIN {X 0,Y 672.584,Z 604.197,A -85,B 0,C 180,E1 31120.639,E2 31120.639} C_VEL
LIN {X 0,Y 672.583,Z 604.198,A -85,B 0,C 180,E1 31117.538,E2 31117.538} C_VEL
LIN {X 0,Y 672.579,Z 604.199,A -85,B 0,C 180,E1 31114.366,E2 31114.366} C_VEL
LIN {X 0,Y 672.583,Z 604.199,A -85,B 0,C 180,E1 31111.293,E2 31111.293} C_VEL
LIN {X 0,Y 672.583,Z 604.198,A -85,B 0,C 180,E1 31108.146,E2 31108.146} C_VEL
LIN {X 0,Y 672.574,Z 604.199,A -85,B 0,C 180,E1 31106.49,E2 31106.49} C_VEL
LIN {X 0,Y 671.602,Z 604.324,A -85,B 0,C 180,E1 31105.834,E2 31105.834} C_VEL
LIN {X 0,Y 665.155,Z 605.129,A -85,B 0,C 180,E1 31103.996,E2 31103.996} C_VEL
LIN {X 0,Y 664.628,Z 605.191,A -85,B 0,C 180,E1 31103.517,E2 31103.517} C_VEL
LIN {X 0,Y 664.641,Z 605.192,A -85,B 0,C 180,E1 31100.509,E2 31100.509} C_VEL
LIN {X 0,Y 664.634,Z 605.181,A -85,B 0,C 180,E1 31097.488,E2 31097.488} C_VEL
LIN {X 0,Y 664.647,Z 605.19,A -85,B 0,C 180,E1 31094.509,E2 31094.509} C_VEL
LIN {X 0,Y 664.652,Z 605.181,A -85,B 0,C 180,E1 31091.35,E2 31091.35} C_VEL
LIN {X 0,Y 664.64,Z 605.19,A -85,B 0,C 180,E1 31088.251,E2 31088.251} C_VEL
LIN {X 0,Y 664.651,Z 605.191,A -85,B 0,C 180,E1 31085.076,E2 31085.076} C_VEL
LIN {X 0,Y 664.635,Z 605.195,A -85,B 0,C 180,E1 31081.951,E2 31081.951} C_VEL
LIN {X 0,Y 664.666,Z 605.377,A -85,B 0,C 180,E1 31081.062,E2 31081.062} C_VEL
LIN {X 0,Y 670.247,Z 623.918,A -85,B 0,C 180,E1 31079.638,E2 31079.638} C_VEL
LIN {X 0,Y 669.893,Z 662.03,A -85,B 0,C 180,E1 31077.127,E2 31077.127} C_VEL
LIN {X 0,Y 669.038,Z 706.08,A -85,B 0,C 180,E1 31074.172,E2 31074.172} C_VEL
LIN {X 0,Y 668.14,Z 751.479,A -85,B 0,C 180,E1 31071.139,E2 31071.139} C_VEL
LIN {X 0,Y 667.35,Z 787.137,A -85,B 0,C 180,E1 31068.75,E2 31068.75} C_VEL
LIN {X 0,Y 666.529,Z 832.117,A -85,B 0,C 180,E1 31065.785,E2 31065.785} C_VEL
LIN {X 0,Y 667.457,Z 842.273,A -85,B 0,C 180,E1 31065.648,E2 31065.648} C_VEL
LIN {X 0,Y 666.709,Z 1001.567,A -85,B 0,C 180,E1 31063.891,E2 31063.891} C_VEL
LIN {X 0,Y 666.517,Z 1018.989,A -85,B 0,C 180,E1 31063.542,E2 31063.542} C_VEL
LIN {X 0,Y 666.214,Z 1035.844,A -85,B 0,C 180,E1 31063.033,E2 31063.033} C_VEL
LIN {X 0,Y 665.843,Z 1052.472,A -85,B 0,C 180,E1 31062.355,E2 31062.355} C_VEL
LIN {X 0,Y 665.469,Z 1067.342,A -85,B 0,C 180,E1 31061.576,E2 31061.576} C_VEL
LIN {X 0,Y 665.08,Z 1081.368,A -85,B 0,C 180,E1 31060.655,E2 31060.655} C_VEL
LIN {X 0,Y 664.704,Z 1095.308,A -85,B 0,C 180,E1 31059.523,E2 31059.523} C_VEL
LIN {X 0,Y 664.434,Z 1106.802,A -85,B 0,C 180,E1 31058.392,E2 31058.392} C_VEL
LIN {X 0,Y 664.224,Z 1116.869,A -85,B 0,C 180,E1 31057.176,E2 31057.176} C_VEL
LIN {X 0,Y 664.066,Z 1126.04,A -85,B 0,C 180,E1 31055.789,E2 31055.789} C_VEL
LIN {X 0,Y 663.98,Z 1133.183,A -85,B 0,C 180,E1 31054.403,E2 31054.403} C_VEL
LIN {X 0,Y 663.936,Z 1138.806,A -85,B 0,C 180,E1 31052.934,E2 31052.934} C_VEL
LIN {X 0,Y 663.917,Z 1142.528,A -85,B 0,C 180,E1 31051.466,E2 31051.466} C_VEL
LIN {X 0,Y 663.924,Z 1144.609,A -85,B 0,C 180,E1 31049.913,E2 31049.913} C_VEL
LIN {X 0,Y 663.914,Z 1144.852,A -85,B 0,C 180,E1 31048.359,E2 31048.359} C_VEL
LIN {X 0,Y 663.919,Z 1143.316,A -85,B 0,C 180,E1 31046.874,E2 31046.874} C_VEL
LIN {X 0,Y 663.927,Z 1139.849,A -85,B 0,C 180,E1 31045.334,E2 31045.334} C_VEL
LIN {X 0,Y 663.965,Z 1134.706,A -85,B 0,C 180,E1 31043.861,E2 31043.861} C_VEL
LIN {X 0,Y 664.041,Z 1128.062,A -85,B 0,C 180,E1 31042.471,E2 31042.471} C_VEL
LIN {X 0,Y 664.178,Z 1119.35,A -85,B 0,C 180,E1 31041.079,E2 31041.079} C_VEL
LIN {X 0,Y 664.38,Z 1109.03,A -85,B 0,C 180,E1 31039.77,E2 31039.77} C_VEL
LIN {X 0,Y 664.639,Z 1098.017,A -85,B 0,C 180,E1 31038.633,E2 31038.633} C_VEL
LIN {X 0,Y 664.994,Z 1084.562,A -85,B 0,C 180,E1 31037.494,E2 31037.494} C_VEL
LIN {X 0,Y 665.38,Z 1070.537,A -85,B 0,C 180,E1 31036.53,E2 31036.53} C_VEL
LIN {X 0,Y 665.773,Z 1055.461,A -85,B 0,C 180,E1 31035.696,E2 31035.696} C_VEL
LIN {X 0,Y 666.124,Z 1040.291,A -85,B 0,C 180,E1 31035.037,E2 31035.037} C_VEL
LIN {X 0,Y 666.441,Z 1023.4,A -85,B 0,C 180,E1 31034.487,E2 31034.487} C_VEL
LIN {X 0,Y 666.671,Z 1005.752,A -85,B 0,C 180,E1 31034.088,E2 31034.088} C_VEL
LIN {X 0,Y 666.81,Z 985.349,A -85,B 0,C 180,E1 31033.82,E2 31033.82} C_VEL
LIN {X 0,Y 667.257,Z 838.072,A -85,B 0,C 180,E1 31032.211,E2 31032.211} C_VEL
LIN {X 0,Y 666.528,Z 831.869,A -85,B 0,C 180,E1 31032.111,E2 31032.111} C_VEL
LIN {X 0,Y 667.347,Z 789.335,A -85,B 0,C 180,E1 31029.291,E2 31029.291} C_VEL
LIN {X 0,Y 668.06,Z 755.74,A -85,B 0,C 180,E1 31027.051,E2 31027.051} C_VEL
LIN {X 0,Y 668.979,Z 708.906,A -85,B 0,C 180,E1 31023.932,E2 31023.932} C_VEL
LIN {X 0,Y 669.866,Z 664.301,A -85,B 0,C 180,E1 31020.93,E2 31020.93} C_VEL
LIN {X 0,Y 670.288,Z 625.668,A -85,B 0,C 180,E1 31018.375,E2 31018.375} C_VEL
LIN {X 0,Y 669.866,Z 622.329,A -85,B 0,C 180,E1 31018.139,E2 31018.139} C_VEL
LIN {X 0,Y 664.651,Z 605.183,A -85,B 0,C 180,E1 31016.797,E2 31016.797} C_VEL
LIN {X 0,Y 664.642,Z 605.182,A -85,B 0,C 180,E1 31013.648,E2 31013.648} C_VEL
LIN {X 0,Y 664.65,Z 605.175,A -85,B 0,C 180,E1 31010.479,E2 31010.479} C_VEL
LIN {X 0,Y 664.647,Z 605.193,A -85,B 0,C 180,E1 31007.362,E2 31007.362} C_VEL
LIN {X 0,Y 664.644,Z 605.184,A -85,B 0,C 180,E1 31004.143,E2 31004.143} C_VEL
LIN {X 0,Y 664.642,Z 605.189,A -85,B 0,C 180,E1 31000.955,E2 31000.955} C_VEL
LIN {X 0,Y 664.651,Z 605.189,A -85,B 0,C 180,E1 30997.832,E2 30997.832} C_VEL
LIN {X 0,Y 664.637,Z 605.19,A -85,B 0,C 180,E1 30994.658,E2 30994.658} C_VEL
LIN {X 0,Y 664.651,Z 605.194,A -85,B 0,C 180,E1 30991.569,E2 30991.569} C_VEL
LIN {X 0,Y 664.645,Z 605.198,A -85,B 0,C 180,E1 30990.764,E2 30990.764} C_VEL
LIN {X 0,Y 665.092,Z 607.009,A -85,B 0,C 180,E1 30990.595,E2 30990.595} C_VEL
LIN {X 0,Y 676.211,Z 626.098,A -85,B 0,C 180,E1 30989.69,E2 30989.69} C_VEL
LIN {X 0,Y 677.184,Z 628.38,A -85,B 0,C 180,E1 30989.607,E2 30989.607} C_VEL
LIN {X 0,Y 674.952,Z 871.333,A -85,B 0,C 180,E1 30986.75,E2 30986.75} C_VEL
LIN {X 0,Y 674.227,Z 946.266,A -85,B 0,C 180,E1 30985.86,E2 30985.86} C_VEL
LIN {X 0,Y 673.771,Z 968.774,A -85,B 0,C 180,E1 30985.467,E2 30985.467} C_VEL
LIN {X 0,Y 673.025,Z 992.293,A -85,B 0,C 180,E1 30984.886,E2 30984.886} C_VEL
LIN {X 0,Y 672.349,Z 1011.869,A -85,B 0,C 180,E1 30984.268,E2 30984.268} C_VEL
LIN {X 0,Y 671.625,Z 1029.379,A -85,B 0,C 180,E1 30983.608,E2 30983.608} C_VEL
LIN {X 0,Y 670.884,Z 1046.718,A -85,B 0,C 180,E1 30982.846,E2 30982.846} C_VEL
LIN {X 0,Y 669.972,Z 1066.057,A -85,B 0,C 180,E1 30981.861,E2 30981.861} C_VEL
LIN {X 0,Y 668.915,Z 1087.563,A -85,B 0,C 180,E1 30980.566,E2 30980.566} C_VEL
LIN {X 0,Y 668.027,Z 1104.737,A -85,B 0,C 180,E1 30979.362,E2 30979.362} C_VEL
LIN {X 0,Y 667.292,Z 1119.907,A -85,B 0,C 180,E1 30978.16,E2 30978.16} C_VEL
LIN {X 0,Y 666.564,Z 1134.795,A -85,B 0,C 180,E1 30976.829,E2 30976.829} C_VEL
LIN {X 0,Y 665.871,Z 1150.457,A -85,B 0,C 180,E1 30975.235,E2 30975.235} C_VEL
LIN {X 0,Y 665.222,Z 1166.043,A -85,B 0,C 180,E1 30973.384,E2 30973.384} C_VEL
LIN {X 0,Y 664.78,Z 1178.13,A -85,B 0,C 180,E1 30971.715,E2 30971.715} C_VEL
LIN {X 0,Y 664.474,Z 1188.032,A -85,B 0,C 180,E1 30970.14,E2 30970.14} C_VEL
LIN {X 0,Y 664.241,Z 1197.501,A -85,B 0,C 180,E1 30968.396,E2 30968.396} C_VEL
LIN {X 0,Y 664.065,Z 1206.816,A -85,B 0,C 180,E1 30966.311,E2 30966.311} C_VEL
LIN {X 0,Y 663.973,Z 1213.758,A -85,B 0,C 180,E1 30964.318,E2 30964.318} C_VEL
LIN {X 0,Y 663.936,Z 1218.194,A -85,B 0,C 180,E1 30962.676,E2 30962.676} C_VEL
LIN {X 0,Y 663.919,Z 1221.671,A -85,B 0,C 180,E1 30960.949,E2 30960.949} C_VEL
LIN {X 0,Y 663.913,Z 1224.143,A -85,B 0,C 180,E1 30958.964,E2 30958.964} C_VEL
LIN {X 0,Y 663.911,Z 1224.951,A -85,B 0,C 180,E1 30956.806,E2 30956.806} C_VEL
LIN {X 0,Y 663.913,Z 1224.081,A -85,B 0,C 180,E1 30954.902,E2 30954.902} C_VEL
LIN {X 0,Y 663.913,Z 1221.704,A -85,B 0,C 180,E1 30952.977,E2 30952.977} C_VEL
LIN {X 0,Y 663.931,Z 1218.063,A -85,B 0,C 180,E1 30951.164,E2 30951.164} C_VEL
LIN {X 0,Y 663.984,Z 1212.126,A -85,B 0,C 180,E1 30949.062,E2 30949.062} C_VEL
LIN {X 0,Y 664.082,Z 1204.855,A -85,B 0,C 180,E1 30947.124,E2 30947.124} C_VEL
LIN {X 0,Y 664.259,Z 1196.21,A -85,B 0,C 180,E1 30945.262,E2 30945.262} C_VEL
LIN {X 0,Y 664.513,Z 1186.851,A -85,B 0,C 180,E1 30943.568,E2 30943.568} C_VEL
LIN {X 0,Y 664.935,Z 1174.003,A -85,B 0,C 180,E1 30941.592,E2 30941.592} C_VEL
LIN {X 0,Y 665.431,Z 1160.8,A -85,B 0,C 180,E1 30939.873,E2 30939.873} C_VEL
LIN {X 0,Y 665.964,Z 1147.994,A -85,B 0,C 180,E1 30938.417,E2 30938.417} C_VEL
LIN {X 0,Y 666.581,Z 1134.395,A -85,B 0,C 180,E1 30937.045,E2 30937.045} C_VEL
LIN {X 0,Y 667.423,Z 1117.323,A -85,B 0,C 180,E1 30935.526,E2 30935.526} C_VEL
LIN {X 0,Y 668.402,Z 1097.716,A -85,B 0,C 180,E1 30934.036,E2 30934.036} C_VEL
LIN {X 0,Y 669.248,Z 1080.383,A -85,B 0,C 180,E1 30932.891,E2 30932.891} C_VEL
LIN {X 0,Y 670.083,Z 1063.517,A -85,B 0,C 180,E1 30931.915,E2 30931.915} C_VEL
LIN {X 0,Y 670.964,Z 1045.114,A -85,B 0,C 180,E1 30930.988,E2 30930.988} C_VEL
LIN {X 0,Y 671.913,Z 1023.232,A -85,B 0,C 180,E1 30930.048,E2 30930.048} C_VEL
LIN {X 0,Y 672.759,Z 1000.737,A -85,B 0,C 180,E1 30929.276,E2 30929.276} C_VEL
LIN {X 0,Y 673.366,Z 981.835,A -85,B 0,C 180,E1 30928.749,E2 30928.749} C_VEL
LIN {X 0,Y 673.876,Z 962.995,A -85,B 0,C 180,E1 30928.333,E2 30928.333} C_VEL
LIN {X 0,Y 674.256,Z 944.428,A -85,B 0,C 180,E1 30928.025,E2 30928.025} C_VEL
LIN {X 0,Y 675.81,Z 759.448,A -85,B 0,C 180,E1 30925.872,E2 30925.872} C_VEL
LIN {X 0,Y 676.086,Z 627.341,A -85,B 0,C 180,E1 30924.432,E2 30924.432} C_VEL
LIN {X 0,Y 669.456,Z 616.85,A -85,B 0,C 180,E1 30924.087,E2 30924.087} C_VEL
LIN {X 0,Y 668.905,Z 615.919,A -85,B 0,C 180,E1 30923.171,E2 30923.171} C_VEL
LIN {X 0,Y 669.324,Z 616.677,A -85,B 0,C 180,E1 30921.932,E2 30921.932} C_VEL
LIN {X 0,Y 670.218,Z 619.297,A -85,B 0,C 180,E1 30920.741,E2 30920.741} C_VEL
LIN {X 0,Y 671.266,Z 621.958,A -85,B 0,C 180,E1 30919.947,E2 30919.947} C_VEL
LIN {X 0,Y 672.822,Z 626.061,A -85,B 0,C 180,E1 30919.052,E2 30919.052} C_VEL
LIN {X 0,Y 669.787,Z 636.918,A -85,B 0,C 180,E1 30918.026,E2 30918.026} C_VEL
LIN {X 0,Y 667.582,Z 649.558,A -85,B 0,C 180,E1 30917.04,E2 30917.04} C_VEL
LIN {X 0,Y 665.985,Z 666.614,A -85,B 0,C 180,E1 30915.924,E2 30915.924} C_VEL
LIN {X 0,Y 664.935,Z 691.381,A -85,B 0,C 180,E1 30914.539,E2 30914.539} C_VEL
LIN {X 0,Y 664.2,Z 743.926,A -85,B 0,C 180,E1 30911.899,E2 30911.899} C_VEL
LIN {X 0,Y 664.937,Z 775.708,A -85,B 0,C 180,E1 30910.324,E2 30910.324} C_VEL
LIN {X 0,Y 667.444,Z 795.412,A -85,B 0,C 180,E1 30909.324,E2 30909.324} C_VEL
LIN {X 0,Y 671.262,Z 810.349,A -85,B 0,C 180,E1 30908.553,E2 30908.553} C_VEL
LIN {X 0,Y 676.823,Z 823.924,A -85,B 0,C 180,E1 30907.848,E2 30907.848} C_VEL
LIN {X 0,Y 683.792,Z 835.801,A -85,B 0,C 180,E1 30907.23,E2 30907.23} C_VEL
LIN {X 0,Y 692.106,Z 846.205,A -85,B 0,C 180,E1 30906.696,E2 30906.696} C_VEL
LIN {X 0,Y 701.655,Z 855.277,A -85,B 0,C 180,E1 30906.237,E2 30906.237} C_VEL
LIN {X 0,Y 707.954,Z 859.94,A -85,B 0,C 180,E1 30905.973,E2 30905.973} C_VEL
LIN {X 0,Y 712.848,Z 862.378,A -85,B 0,C 180,E1 30905.693,E2 30905.693} C_VEL
LIN {X 0,Y 717.894,Z 863.66,A -85,B 0,C 180,E1 30905.295,E2 30905.295} C_VEL
LIN {X 0,Y 721.616,Z 863.494,A -85,B 0,C 180,E1 30904.886,E2 30904.886} C_VEL
LIN {X 0,Y 724.219,Z 862.252,A -85,B 0,C 180,E1 30904.477,E2 30904.477} C_VEL
LIN {X 0,Y 725.921,Z 859.718,A -85,B 0,C 180,E1 30904.003,E2 30904.003} C_VEL
LIN {X 0,Y 726.121,Z 856.079,A -85,B 0,C 180,E1 30903.542,E2 30903.542} C_VEL
LIN {X 0,Y 724.75,Z 851.699,A -85,B 0,C 180,E1 30903.14,E2 30903.14} C_VEL
LIN {X 0,Y 719.586,Z 841.315,A -85,B 0,C 180,E1 30902.484,E2 30902.484} C_VEL
LIN {X 0,Y 716.134,Z 832.861,A -85,B 0,C 180,E1 30902.048,E2 30902.048} C_VEL
LIN {X 0,Y 712.183,Z 875.076,A -85,B 0,C 180,E1 30901.536,E2 30901.536} C_VEL
LIN {X 0,Y 709.644,Z 892.377,A -85,B 0,C 180,E1 30901.281,E2 30901.281} C_VEL
LIN {X 0,Y 706.71,Z 903.653,A -85,B 0,C 180,E1 30901.052,E2 30901.052} C_VEL
LIN {X 0,Y 705.886,Z 906.58,A -85,B 0,C 180,E1 30901.005,E2 30901.005} C_VEL
LIN {X 0,Y 701.447,Z 920.023,A -85,B 0,C 180,E1 30900.971,E2 30900.971} C_VEL
LIN {X 0,Y 695.349,Z 932.754,A -85,B 0,C 180,E1 30900.888,E2 30900.888} C_VEL
LIN {X 0,Y 689.009,Z 943.936,A -85,B 0,C 180,E1 30900.685,E2 30900.685} C_VEL
LIN {X 0,Y 684.13,Z 952.977,A -85,B 0,C 180,E1 30900.378,E2 30900.378} C_VEL
LIN {X 0,Y 681.347,Z 958.753,A -85,B 0,C 180,E1 30900.126,E2 30900.126} C_VEL
LIN {X 0,Y 677.634,Z 966.065,A -85,B 0,C 180,E1 30899.815,E2 30899.815} C_VEL
LIN {X 0,Y 674.675,Z 973.831,A -85,B 0,C 180,E1 30899.419,E2 30899.419} C_VEL
LIN {X 0,Y 674.195,Z 1019.475,A -85,B 0,C 180,E1 30898.863,E2 30898.863} C_VEL
LIN {X 0,Y 673.646,Z 1042.555,A -85,B 0,C 180,E1 30898.431,E2 30898.431} C_VEL
LIN {X 0,Y 672.949,Z 1065.544,A -85,B 0,C 180,E1 30897.84,E2 30897.84} C_VEL
LIN {X 0,Y 672.164,Z 1087.278,A -85,B 0,C 180,E1 30897.126,E2 30897.126} C_VEL
LIN {X 0,Y 671.199,Z 1109.822,A -85,B 0,C 180,E1 30896.213,E2 30896.213} C_VEL
LIN {X 0,Y 670.219,Z 1131.319,A -85,B 0,C 180,E1 30895.163,E2 30895.163} C_VEL
LIN {X 0,Y 669.181,Z 1152.253,A -85,B 0,C 180,E1 30893.951,E2 30893.951} C_VEL
LIN {X 0,Y 668.171,Z 1172.449,A -85,B 0,C 180,E1 30892.584,E2 30892.584} C_VEL
LIN {X 0,Y 667.166,Z 1192.588,A -85,B 0,C 180,E1 30890.98,E2 30890.98} C_VEL
LIN {X 0,Y 666.419,Z 1207.961,A -85,B 0,C 180,E1 30889.567,E2 30889.567} C_VEL
LIN {X 0,Y 665.782,Z 1222.279,A -85,B 0,C 180,E1 30888.073,E2 30888.073} C_VEL
LIN {X 0,Y 665.226,Z 1236.173,A -85,B 0,C 180,E1 30886.415,E2 30886.415} C_VEL
LIN {X 0,Y 664.717,Z 1250.133,A -85,B 0,C 180,E1 30884.461,E2 30884.461} C_VEL
LIN {X 0,Y 664.413,Z 1260.372,A -85,B 0,C 180,E1 30882.782,E2 30882.782} C_VEL
LIN {X 0,Y 664.18,Z 1269.962,A -85,B 0,C 180,E1 30880.936,E2 30880.936} C_VEL
LIN {X 0,Y 664.018,Z 1278.795,A -85,B 0,C 180,E1 30878.836,E2 30878.836} C_VEL
LIN {X 0,Y 663.947,Z 1284.823,A -85,B 0,C 180,E1 30877.008,E2 30877.008} C_VEL
LIN {X 0,Y 663.926,Z 1289.244,A -85,B 0,C 180,E1 30875.272,E2 30875.272} C_VEL
LIN {X 0,Y 663.906,Z 1292.769,A -85,B 0,C 180,E1 30873.282,E2 30873.282} C_VEL
LIN {X 0,Y 663.904,Z 1294.662,A -85,B 0,C 180,E1 30871.209,E2 30871.209} C_VEL
LIN {X 0,Y 663.893,Z 1294.85,A -85,B 0,C 180,E1 30869.397,E2 30869.397} C_VEL
LIN {X 0,Y 663.898,Z 1293.746,A -85,B 0,C 180,E1 30867.584,E2 30867.584} C_VEL
LIN {X 0,Y 663.907,Z 1290.998,A -85,B 0,C 180,E1 30865.596,E2 30865.596} C_VEL
LIN {X 0,Y 663.937,Z 1286.324,A -85,B 0,C 180,E1 30863.516,E2 30863.516} C_VEL
LIN {X 0,Y 664.009,Z 1280.657,A -85,B 0,C 180,E1 30861.689,E2 30861.689} C_VEL
LIN {X 0,Y 664.103,Z 1273.877,A -85,B 0,C 180,E1 30859.943,E2 30859.943} C_VEL
LIN {X 0,Y 664.311,Z 1264.735,A -85,B 0,C 180,E1 30858.013,E2 30858.013} C_VEL
LIN {X 0,Y 664.628,Z 1253.207,A -85,B 0,C 180,E1 30856.017,E2 30856.017} C_VEL
LIN {X 0,Y 664.978,Z 1242.154,A -85,B 0,C 180,E1 30854.388,E2 30854.388} C_VEL
LIN {X 0,Y 665.475,Z 1229.694,A -85,B 0,C 180,E1 30852.784,E2 30852.784} C_VEL
LIN {X 0,Y 666.182,Z 1213.646,A -85,B 0,C 180,E1 30850.993,E2 30850.993} C_VEL
LIN {X 0,Y 666.916,Z 1197.261,A -85,B 0,C 180,E1 30849.432,E2 30849.432} C_VEL
LIN {X 0,Y 667.681,Z 1182.057,A -85,B 0,C 180,E1 30848.154,E2 30848.154} C_VEL
LIN {X 0,Y 668.578,Z 1164.33,A -85,B 0,C 180,E1 30846.84,E2 30846.84} C_VEL
LIN {X 0,Y 669.583,Z 1144.361,A -85,B 0,C 180,E1 30845.568,E2 30845.568} C_VEL
LIN {X 0,Y 670.571,Z 1123.597,A -85,B 0,C 180,E1 30844.438,E2 30844.438} C_VEL
LIN {X 0,Y 671.557,Z 1101.872,A -85,B 0,C 180,E1 30843.444,E2 30843.444} C_VEL
LIN {X 0,Y 672.449,Z 1079.532,A -85,B 0,C 180,E1 30842.601,E2 30842.601} C_VEL
LIN {X 0,Y 673.244,Z 1056.652,A -85,B 0,C 180,E1 30841.912,E2 30841.912} C_VEL
LIN {X 0,Y 673.897,Z 1033.644,A -85,B 0,C 180,E1 30841.384,E2 30841.384} C_VEL
LIN {X 0,Y 674.352,Z 1009.527,A -85,B 0,C 180,E1 30840.996,E2 30840.996} C_VEL
LIN {X 0,Y 674.68,Z 973.426,A -85,B 0,C 180,E1 30840.576,E2 30840.576} C_VEL
LIN {X 0,Y 679.176,Z 962.746,A -85,B 0,C 180,E1 30840.028,E2 30840.028} C_VEL
LIN {X 0,Y 682.8,Z 955.86,A -85,B 0,C 180,E1 30839.753,E2 30839.753} C_VEL
LIN {X 0,Y 686.867,Z 947.737,A -85,B 0,C 180,E1 30839.426,E2 30839.426} C_VEL
LIN {X 0,Y 692.808,Z 937.32,A -85,B 0,C 180,E1 30839.175,E2 30839.175} C_VEL
LIN {X 0,Y 699.248,Z 925.047,A -85,B 0,C 180,E1 30839.05,E2 30839.05} C_VEL
LIN {X 0,Y 704.407,Z 911.804,A -85,B 0,C 180,E1 30839.008,E2 30839.008} C_VEL
LIN {X 0,Y 706.483,Z 904.371,A -85,B 0,C 180,E1 30838.969,E2 30838.969} C_VEL
LIN {X 0,Y 709.383,Z 893.592,A -85,B 0,C 180,E1 30838.739,E2 30838.739} C_VEL
LIN {X 0,Y 711.956,Z 877.161,A -85,B 0,C 180,E1 30838.493,E2 30838.493} C_VEL
LIN {X 0,Y 715.855,Z 836.193,A -85,B 0,C 180,E1 30837.988,E2 30837.988} C_VEL
LIN {X 0,Y 716.235,Z 832.843,A -85,B 0,C 180,E1 30837.939,E2 30837.939} C_VEL
LIN {X 0,Y 720.985,Z 844.354,A -85,B 0,C 180,E1 30837.342,E2 30837.342} C_VEL
LIN {X 0,Y 725.088,Z 852.48,A -85,B 0,C 180,E1 30836.797,E2 30836.797} C_VEL
LIN {X 0,Y 726.199,Z 856.776,A -85,B 0,C 180,E1 30836.382,E2 30836.382} C_VEL
LIN {X 0,Y 725.927,Z 859.699,A -85,B 0,C 180,E1 30836,E2 30836} C_VEL
LIN {X 0,Y 724.186,Z 862.278,A -85,B 0,C 180,E1 30835.516,E2 30835.516} C_VEL
LIN {X 0,Y 721.04,Z 863.607,A -85,B 0,C 180,E1 30835.041,E2 30835.041} C_VEL
LIN {X 0,Y 717.217,Z 863.573,A -85,B 0,C 180,E1 30834.644,E2 30834.644} C_VEL
LIN {X 0,Y 712.102,Z 862.107,A -85,B 0,C 180,E1 30834.252,E2 30834.252} C_VEL
LIN {X 0,Y 702.651,Z 857.65,A -85,B 0,C 180,E1 30833.502,E2 30833.502} C_VEL
LIN {X 0,Y 694.196,Z 851.651,A -85,B 0,C 180,E1 30832.663,E2 30832.663} C_VEL
LIN {X 0,Y 687.267,Z 844.366,A -85,B 0,C 180,E1 30831.78,E2 30831.78} C_VEL
LIN {X 0,Y 681.683,Z 835.408,A -85,B 0,C 180,E1 30830.817,E2 30830.817} C_VEL
LIN {X 0,Y 677.611,Z 824.777,A -85,B 0,C 180,E1 30829.785,E2 30829.785} C_VEL
LIN {X 0,Y 675.273,Z 812.577,A -85,B 0,C 180,E1 30828.711,E2 30828.711} C_VEL
LIN {X 0,Y 674.588,Z 795.873,A -85,B 0,C 180,E1 30827.363,E2 30827.363} C_VEL
LIN {X 0,Y 676.256,Z 755.735,A -85,B 0,C 180,E1 30824.258,E2 30824.258} C_VEL
LIN {X 0,Y 677.839,Z 719.038,A -85,B 0,C 180,E1 30821.34,E2 30821.34} C_VEL
LIN {X 0,Y 679.314,Z 684.447,A -85,B 0,C 180,E1 30818.508,E2 30818.508} C_VEL
LIN {X 0,Y 680.757,Z 650.241,A -85,B 0,C 180,E1 30815.618,E2 30815.618} C_VEL
LIN {X 0,Y 680.941,Z 642.959,A -85,B 0,C 180,E1 30814.982,E2 30814.982} C_VEL
LIN {X 0,Y 672.198,Z 622.82,A -85,B 0,C 180,E1 30812.343,E2 30812.343} C_VEL
LIN {X 0,Y 665.969,Z 608.723,A -85,B 0,C 180,E1 30810.396,E2 30810.396} C_VEL
LIN {X 0,Y 664.635,Z 605.194,A -85,B 0,C 180,E1 30809.882,E2 30809.882} C_VEL
LIN {X 0,Y 664.635,Z 605.193,A -85,B 0,C 180,E1 30806.829,E2 30806.829} C_VEL
LIN {X 0,Y 664.629,Z 605.193,A -85,B 0,C 180,E1 30803.778,E2 30803.778} C_VEL
LIN {X 0,Y 664.636,Z 605.19,A -85,B 0,C 180,E1 30800.796,E2 30800.796} C_VEL
LIN {X 0,Y 664.631,Z 605.192,A -85,B 0,C 180,E1 30797.774,E2 30797.774} C_VEL
LIN {X 0,Y 664.649,Z 605.19,A -85,B 0,C 180,E1 30794.729,E2 30794.729} C_VEL
LIN {X 0,Y 664.644,Z 605.193,A -85,B 0,C 180,E1 30791.63,E2 30791.63} C_VEL
LIN {X 0,Y 664.643,Z 605.19,A -85,B 0,C 180,E1 30788.565,E2 30788.565} C_VEL
LIN {X 0,Y 664.651,Z 605.188,A -85,B 0,C 180,E1 30785.438,E2 30785.438} C_VEL
LIN {X 0,Y 664.638,Z 605.192,A -85,B 0,C 180,E1 30782.328,E2 30782.328} C_VEL
LIN {X 0,Y 664.648,Z 605.19,A -85,B 0,C 180,E1 30779.224,E2 30779.224} C_VEL
LIN {X 0,Y 664.636,Z 605.191,A -85,B 0,C 180,E1 30776.118,E2 30776.118} C_VEL
LIN {X 0,Y 664.644,Z 605.188,A -85,B 0,C 180,E1 30773.001,E2 30773.001} C_VEL
LIN {X 0,Y 664.639,Z 605.187,A -85,B 0,C 180,E1 30769.95,E2 30769.95} C_VEL
LIN {X 0,Y 664.645,Z 605.185,A -85,B 0,C 180,E1 30766.87,E2 30766.87} C_VEL
LIN {X 0,Y 664.64,Z 605.186,A -85,B 0,C 180,E1 30763.75,E2 30763.75} C_VEL
LIN {X 0,Y 664.643,Z 605.187,A -85,B 0,C 180,E1 30760.581,E2 30760.581} C_VEL
LIN {X 0,Y 664.638,Z 605.188,A -85,B 0,C 180,E1 30757.441,E2 30757.441} C_VEL
LIN {X 0,Y 664.638,Z 605.188,A -85,B 0,C 180,E1 30754.304,E2 30754.304} C_VEL
LIN {X 0,Y 664.639,Z 605.188,A -85,B 0,C 180,E1 30751.222,E2 30751.222} C_VEL
LIN {X 0,Y 664.643,Z 605.187,A -85,B 0,C 180,E1 30748.126,E2 30748.126} C_VEL
LIN {X 0,Y 664.638,Z 605.185,A -85,B 0,C 180,E1 30745.027,E2 30745.027} C_VEL
LIN {X 0,Y 664.628,Z 605.191,A -85,B 0,C 180,E1 30743.517,E2 30743.517} C_VEL
LIN {X 0,Y 663.655,Z 605.313,A -85,B 0,C 180,E1 30742.853,E2 30742.853} C_VEL
LIN {X 0,Y 657.244,Z 606.117,A -85,B 0,C 180,E1 30740.992,E2 30740.992} C_VEL
LIN {X 0,Y 656.702,Z 606.181,A -85,B 0,C 180,E1 30740.508,E2 30740.508} C_VEL
LIN {X 0,Y 656.694,Z 606.169,A -85,B 0,C 180,E1 30737.465,E2 30737.465} C_VEL
LIN {X 0,Y 656.709,Z 606.18,A -85,B 0,C 180,E1 30734.431,E2 30734.431} C_VEL
LIN {X 0,Y 656.713,Z 606.169,A -85,B 0,C 180,E1 30731.355,E2 30731.355} C_VEL
LIN {X 0,Y 656.7,Z 606.178,A -85,B 0,C 180,E1 30728.218,E2 30728.218} C_VEL
LIN {X 0,Y 656.712,Z 606.18,A -85,B 0,C 180,E1 30725.135,E2 30725.135} C_VEL
LIN {X 0,Y 656.697,Z 606.184,A -85,B 0,C 180,E1 30721.994,E2 30721.994} C_VEL
LIN {X 0,Y 656.718,Z 606.219,A -85,B 0,C 180,E1 30721.355,E2 30721.355} C_VEL
LIN {X 0,Y 662.797,Z 626.957,A -85,B 0,C 180,E1 30719.755,E2 30719.755} C_VEL
LIN {X 0,Y 662.377,Z 665.27,A -85,B 0,C 180,E1 30717.217,E2 30717.217} C_VEL
LIN {X 0,Y 661.457,Z 709.522,A -85,B 0,C 180,E1 30714.229,E2 30714.229} C_VEL
LIN {X 0,Y 660.462,Z 755.809,A -85,B 0,C 180,E1 30711.118,E2 30711.118} C_VEL
LIN {X 0,Y 659.518,Z 800.279,A -85,B 0,C 180,E1 30708.152,E2 30708.152} C_VEL
LIN {X 0,Y 658.975,Z 833.524,A -85,B 0,C 180,E1 30705.977,E2 30705.977} C_VEL
LIN {X 0,Y 659.821,Z 843.151,A -85,B 0,C 180,E1 30705.846,E2 30705.846} C_VEL
LIN {X 0,Y 659.007,Z 1002.55,A -85,B 0,C 180,E1 30704.068,E2 30704.068} C_VEL
LIN {X 0,Y 658.814,Z 1019.961,A -85,B 0,C 180,E1 30703.715,E2 30703.715} C_VEL
LIN {X 0,Y 658.509,Z 1036.569,A -85,B 0,C 180,E1 30703.209,E2 30703.209} C_VEL
LIN {X 0,Y 658.131,Z 1052.722,A -85,B 0,C 180,E1 30702.547,E2 30702.547} C_VEL
LIN {X 0,Y 657.729,Z 1067.841,A -85,B 0,C 180,E1 30701.753,E2 30701.753} C_VEL
LIN {X 0,Y 657.315,Z 1081.894,A -85,B 0,C 180,E1 30700.827,E2 30700.827} C_VEL
LIN {X 0,Y 656.939,Z 1094.386,A -85,B 0,C 180,E1 30699.814,E2 30699.814} C_VEL
LIN {X 0,Y 656.595,Z 1105.957,A -85,B 0,C 180,E1 30698.67,E2 30698.67} C_VEL
LIN {X 0,Y 656.323,Z 1116.11,A -85,B 0,C 180,E1 30697.439,E2 30697.439} C_VEL
LIN {X 0,Y 656.125,Z 1124.853,A -85,B 0,C 180,E1 30696.122,E2 30696.122} C_VEL
LIN {X 0,Y 655.999,Z 1132.109,A -85,B 0,C 180,E1 30694.72,E2 30694.72} C_VEL
LIN {X 0,Y 655.942,Z 1138.264,A -85,B 0,C 180,E1 30693.145,E2 30693.145} C_VEL
LIN {X 0,Y 655.917,Z 1142.23,A -85,B 0,C 180,E1 30691.659,E2 30691.659} C_VEL
LIN {X 0,Y 655.924,Z 1144.416,A -85,B 0,C 180,E1 30690.173,E2 30690.173} C_VEL
LIN {X 0,Y 655.914,Z 1144.916,A -85,B 0,C 180,E1 30688.601,E2 30688.601} C_VEL
LIN {X 0,Y 655.918,Z 1143.582,A -85,B 0,C 180,E1 30687.028,E2 30687.028} C_VEL
LIN {X 0,Y 655.927,Z 1140.538,A -85,B 0,C 180,E1 30685.53,E2 30685.53} C_VEL
LIN {X 0,Y 655.96,Z 1135.7,A -85,B 0,C 180,E1 30684.049,E2 30684.049} C_VEL
LIN {X 0,Y 656.049,Z 1129.052,A -85,B 0,C 180,E1 30682.555,E2 30682.555} C_VEL
LIN {X 0,Y 656.213,Z 1120.862,A -85,B 0,C 180,E1 30681.146,E2 30681.146} C_VEL
LIN {X 0,Y 656.454,Z 1111.022,A -85,B 0,C 180,E1 30679.822,E2 30679.822} C_VEL
LIN {X 0,Y 656.78,Z 1099.618,A -85,B 0,C 180,E1 30678.584,E2 30678.584} C_VEL
LIN {X 0,Y 657.166,Z 1087.079,A -85,B 0,C 180,E1 30677.477,E2 30677.477} C_VEL
LIN {X 0,Y 657.574,Z 1073.191,A -85,B 0,C 180,E1 30676.488,E2 30676.488} C_VEL
LIN {X 0,Y 657.994,Z 1058.03,A -85,B 0,C 180,E1 30675.621,E2 30675.621} C_VEL
LIN {X 0,Y 658.393,Z 1042.032,A -85,B 0,C 180,E1 30674.902,E2 30674.902} C_VEL
LIN {X 0,Y 658.726,Z 1025.161,A -85,B 0,C 180,E1 30674.338,E2 30674.338} C_VEL
LIN {X 0,Y 658.967,Z 1007.281,A -85,B 0,C 180,E1 30673.923,E2 30673.923} C_VEL
LIN {X 0,Y 659.106,Z 987.559,A -85,B 0,C 180,E1 30673.655,E2 30673.655} C_VEL
LIN {X 0,Y 659.61,Z 838.737,A -85,B 0,C 180,E1 30672.009,E2 30672.009} C_VEL
LIN {X 0,Y 658.907,Z 832.948,A -85,B 0,C 180,E1 30671.92,E2 30671.92} C_VEL
LIN {X 0,Y 659.855,Z 785.493,A -85,B 0,C 180,E1 30668.766,E2 30668.766} C_VEL
LIN {X 0,Y 660.782,Z 739.37,A -85,B 0,C 180,E1 30665.694,E2 30665.694} C_VEL
LIN {X 0,Y 661.827,Z 693.985,A -85,B 0,C 180,E1 30662.627,E2 30662.627} C_VEL
LIN {X 0,Y 662.625,Z 651.109,A -85,B 0,C 180,E1 30659.734,E2 30659.734} C_VEL
LIN {X 0,Y 662.797,Z 626.078,A -85,B 0,C 180,E1 30658.077,E2 30658.077} C_VEL
LIN {X 0,Y 656.698,Z 606.17,A -85,B 0,C 180,E1 30656.499,E2 30656.499} C_VEL
LIN {X 0,Y 656.7,Z 606.17,A -85,B 0,C 180,E1 30653.463,E2 30653.463} C_VEL
LIN {X 0,Y 656.703,Z 606.164,A -85,B 0,C 180,E1 30650.359,E2 30650.359} C_VEL
LIN {X 0,Y 656.709,Z 606.179,A -85,B 0,C 180,E1 30647.213,E2 30647.213} C_VEL
LIN {X 0,Y 656.702,Z 606.174,A -85,B 0,C 180,E1 30644.055,E2 30644.055} C_VEL
LIN {X 0,Y 656.7,Z 606.178,A -85,B 0,C 180,E1 30640.899,E2 30640.899} C_VEL
LIN {X 0,Y 656.711,Z 606.179,A -85,B 0,C 180,E1 30637.794,E2 30637.794} C_VEL
LIN {X 0,Y 656.7,Z 606.18,A -85,B 0,C 180,E1 30634.693,E2 30634.693} C_VEL
LIN {X 0,Y 656.713,Z 606.183,A -85,B 0,C 180,E1 30631.585,E2 30631.585} C_VEL
LIN {X 0,Y 656.73,Z 606.445,A -85,B 0,C 180,E1 30631.278,E2 30631.278} C_VEL
LIN {X 0,Y 657.47,Z 608.758,A -85,B 0,C 180,E1 30631.038,E2 30631.038} C_VEL
LIN {X 0,Y 659.85,Z 612.574,A -85,B 0,C 180,E1 30630.837,E2 30630.837} C_VEL
LIN {X 0,Y 670.313,Z 630.405,A -85,B 0,C 180,E1 30629.969,E2 30629.969} C_VEL
LIN {X 0,Y 668.659,Z 795.762,A -85,B 0,C 180,E1 30627.973,E2 30627.973} C_VEL
LIN {X 0,Y 667.229,Z 945.25,A -85,B 0,C 180,E1 30626.207,E2 30626.207} C_VEL
LIN {X 0,Y 666.804,Z 964.596,A -85,B 0,C 180,E1 30625.877,E2 30625.877} C_VEL
LIN {X 0,Y 666.108,Z 988.056,A -85,B 0,C 180,E1 30625.334,E2 30625.334} C_VEL
LIN {X 0,Y 665.242,Z 1010.051,A -85,B 0,C 180,E1 30624.652,E2 30624.652} C_VEL
LIN {X 0,Y 664.448,Z 1028.123,A -85,B 0,C 180,E1 30623.973,E2 30623.973} C_VEL
LIN {X 0,Y 663.684,Z 1044.664,A -85,B 0,C 180,E1 30623.249,E2 30623.249} C_VEL
LIN {X 0,Y 662.809,Z 1061.809,A -85,B 0,C 180,E1 30622.386,E2 30622.386} C_VEL
LIN {X 0,Y 661.846,Z 1079.706,A -85,B 0,C 180,E1 30621.352,E2 30621.352} C_VEL
LIN {X 0,Y 660.734,Z 1100.454,A -85,B 0,C 180,E1 30619.958,E2 30619.958} C_VEL
LIN {X 0,Y 659.754,Z 1117.719,A -85,B 0,C 180,E1 30618.604,E2 30618.604} C_VEL
LIN {X 0,Y 658.986,Z 1132.364,A -85,B 0,C 180,E1 30617.301,E2 30617.301} C_VEL
LIN {X 0,Y 658.293,Z 1145.798,A -85,B 0,C 180,E1 30615.955,E2 30615.955} C_VEL
LIN {X 0,Y 657.693,Z 1158.459,A -85,B 0,C 180,E1 30614.528,E2 30614.528} C_VEL
LIN {X 0,Y 657.114,Z 1172.358,A -85,B 0,C 180,E1 30612.741,E2 30612.741} C_VEL
LIN {X 0,Y 656.628,Z 1185.141,A -85,B 0,C 180,E1 30610.795,E2 30610.795} C_VEL
LIN {X 0,Y 656.357,Z 1194.54,A -85,B 0,C 180,E1 30609.116,E2 30609.116} C_VEL
LIN {X 0,Y 656.161,Z 1202.544,A -85,B 0,C 180,E1 30607.442,E2 30607.442} C_VEL
LIN {X 0,Y 656.019,Z 1210.007,A -85,B 0,C 180,E1 30605.561,E2 30605.561} C_VEL
LIN {X 0,Y 655.946,Z 1216.428,A -85,B 0,C 180,E1 30603.496,E2 30603.496} C_VEL
LIN {X 0,Y 655.911,Z 1221,A -85,B 0,C 180,E1 30601.398,E2 30601.398} C_VEL
LIN {X 0,Y 655.911,Z 1223.576,A -85,B 0,C 180,E1 30599.563,E2 30599.563} C_VEL
LIN {X 0,Y 655.903,Z 1224.806,A -85,B 0,C 180,E1 30597.728,E2 30597.728} C_VEL
LIN {X 0,Y 655.909,Z 1224.706,A -85,B 0,C 180,E1 30595.891,E2 30595.891} C_VEL
LIN {X 0,Y 655.909,Z 1222.97,A -85,B 0,C 180,E1 30593.786,E2 30593.786} C_VEL
LIN {X 0,Y 655.928,Z 1219.554,A -85,B 0,C 180,E1 30591.762,E2 30591.762} C_VEL
LIN {X 0,Y 655.966,Z 1215.1,A -85,B 0,C 180,E1 30589.966,E2 30589.966} C_VEL
LIN {X 0,Y 656.025,Z 1209.816,A -85,B 0,C 180,E1 30588.304,E2 30588.304} C_VEL
LIN {X 0,Y 656.164,Z 1202.39,A -85,B 0,C 180,E1 30586.428,E2 30586.428} C_VEL
LIN {X 0,Y 656.405,Z 1192.797,A -85,B 0,C 180,E1 30584.449,E2 30584.449} C_VEL
LIN {X 0,Y 656.76,Z 1181.615,A -85,B 0,C 180,E1 30582.547,E2 30582.547} C_VEL
LIN {X 0,Y 657.191,Z 1170.384,A -85,B 0,C 180,E1 30580.906,E2 30580.906} C_VEL
LIN {X 0,Y 657.706,Z 1158.174,A -85,B 0,C 180,E1 30579.347,E2 30579.347} C_VEL
LIN {X 0,Y 658.336,Z 1145.047,A -85,B 0,C 180,E1 30577.873,E2 30577.873} C_VEL
LIN {X 0,Y 659.277,Z 1127.077,A -85,B 0,C 180,E1 30576.112,E2 30576.112} C_VEL
LIN {X 0,Y 660.203,Z 1109.831,A -85,B 0,C 180,E1 30574.669,E2 30574.669} C_VEL
LIN {X 0,Y 661.017,Z 1094.653,A -85,B 0,C 180,E1 30573.546,E2 30573.546} C_VEL
LIN {X 0,Y 661.878,Z 1078.958,A -85,B 0,C 180,E1 30572.515,E2 30572.515} C_VEL
LIN {X 0,Y 662.805,Z 1061.906,A -85,B 0,C 180,E1 30571.529,E2 30571.529} C_VEL
LIN {X 0,Y 663.832,Z 1041.974,A -85,B 0,C 180,E1 30570.53,E2 30570.53} C_VEL
LIN {X 0,Y 664.88,Z 1018.856,A -85,B 0,C 180,E1 30569.574,E2 30569.574} C_VEL
LIN {X 0,Y 665.641,Z 1000.156,A -85,B 0,C 180,E1 30568.936,E2 30568.936} C_VEL
LIN {X 0,Y 666.283,Z 981.818,A -85,B 0,C 180,E1 30568.422,E2 30568.422} C_VEL
LIN {X 0,Y 666.823,Z 963.473,A -85,B 0,C 180,E1 30568.012,E2 30568.012} C_VEL
LIN {X 0,Y 667.237,Z 945.156,A -85,B 0,C 180,E1 30567.703,E2 30567.703} C_VEL
LIN {X 0,Y 667.733,Z 891.713,A -85,B 0,C 180,E1 30567.071,E2 30567.071} C_VEL
LIN {X 0,Y 668.831,Z 630.321,A -85,B 0,C 180,E1 30564.218,E2 30564.218} C_VEL
LIN {X 0,Y 662.992,Z 621.522,A -85,B 0,C 180,E1 30563.912,E2 30563.912} C_VEL
LIN {X 0,Y 662.623,Z 620.908,A -85,B 0,C 180,E1 30562.872,E2 30562.872} C_VEL
LIN {X 0,Y 663.301,Z 622.142,A -85,B 0,C 180,E1 30561.606,E2 30561.606} C_VEL
LIN {X 0,Y 664.625,Z 625.8,A -85,B 0,C 180,E1 30560.244,E2 30560.244} C_VEL
LIN {X 0,Y 666.098,Z 630.096,A -85,B 0,C 180,E1 30559.245,E2 30559.245} C_VEL
LIN {X 0,Y 662.578,Z 641.264,A -85,B 0,C 180,E1 30558.162,E2 30558.162} C_VEL
LIN {X 0,Y 660.07,Z 654.519,A -85,B 0,C 180,E1 30557.09,E2 30557.09} C_VEL
LIN {X 0,Y 658.375,Z 670.795,A -85,B 0,C 180,E1 30555.982,E2 30555.982} C_VEL
LIN {X 0,Y 657.184,Z 694.472,A -85,B 0,C 180,E1 30554.598,E2 30554.598} C_VEL
LIN {X 0,Y 656.342,Z 740.313,A -85,B 0,C 180,E1 30552.209,E2 30552.209} C_VEL
LIN {X 0,Y 656.852,Z 774.192,A -85,B 0,C 180,E1 30550.493,E2 30550.493} C_VEL
LIN {X 0,Y 659.123,Z 794.339,A -85,B 0,C 180,E1 30549.452,E2 30549.452} C_VEL
LIN {X 0,Y 662.879,Z 810.301,A -85,B 0,C 180,E1 30548.615,E2 30548.615} C_VEL
LIN {X 0,Y 668.224,Z 824.191,A -85,B 0,C 180,E1 30547.878,E2 30547.878} C_VEL
LIN {X 0,Y 674.953,Z 836.483,A -85,B 0,C 180,E1 30547.225,E2 30547.225} C_VEL
LIN {X 0,Y 683.014,Z 847.331,A -85,B 0,C 180,E1 30546.655,E2 30546.655} C_VEL
LIN {X 0,Y 692.328,Z 856.966,A -85,B 0,C 180,E1 30546.163,E2 30546.163} C_VEL
LIN {X 0,Y 703.202,Z 865.557,A -85,B 0,C 180,E1 30545.716,E2 30545.716} C_VEL
LIN {X 0,Y 708.354,Z 868.355,A -85,B 0,C 180,E1 30545.464,E2 30545.464} C_VEL
LIN {X 0,Y 713.676,Z 869.988,A -85,B 0,C 180,E1 30545.094,E2 30545.094} C_VEL
LIN {X 0,Y 717.652,Z 870.152,A -85,B 0,C 180,E1 30544.71,E2 30544.71} C_VEL
LIN {X 0,Y 720.985,Z 869.024,A -85,B 0,C 180,E1 30544.253,E2 30544.253} C_VEL
LIN {X 0,Y 723.013,Z 866.678,A -85,B 0,C 180,E1 30543.777,E2 30543.777} C_VEL
LIN {X 0,Y 723.551,Z 863.342,A -85,B 0,C 180,E1 30543.321,E2 30543.321} C_VEL
LIN {X 0,Y 722.537,Z 859.105,A -85,B 0,C 180,E1 30542.9,E2 30542.9} C_VEL
LIN {X 0,Y 718.782,Z 851.976,A -85,B 0,C 180,E1 30542.383,E2 30542.383} C_VEL
LIN {X 0,Y 716.161,Z 875.079,A -85,B 0,C 180,E1 30542.108,E2 30542.108} C_VEL
LIN {X 0,Y 712.389,Z 890.814,A -85,B 0,C 180,E1 30541.937,E2 30541.937} C_VEL
LIN {X 0,Y 708.033,Z 903.284,A -85,B 0,C 180,E1 30541.74,E2 30541.74} C_VEL
LIN {X 0,Y 706.321,Z 907.582,A -85,B 0,C 180,E1 30541.65,E2 30541.65} C_VEL
LIN {X 0,Y 700.029,Z 920.213,A -85,B 0,C 180,E1 30541.616,E2 30541.616} C_VEL
LIN {X 0,Y 692.219,Z 932.222,A -85,B 0,C 180,E1 30541.495,E2 30541.495} C_VEL
LIN {X 0,Y 684.552,Z 942.992,A -85,B 0,C 180,E1 30541.235,E2 30541.235} C_VEL
LIN {X 0,Y 678.851,Z 951.953,A -85,B 0,C 180,E1 30540.885,E2 30540.885} C_VEL
LIN {X 0,Y 675.099,Z 958.851,A -85,B 0,C 180,E1 30540.561,E2 30540.561} C_VEL
LIN {X 0,Y 670.855,Z 966.717,A -85,B 0,C 180,E1 30540.177,E2 30540.177} C_VEL
LIN {X 0,Y 667.645,Z 975.023,A -85,B 0,C 180,E1 30539.735,E2 30539.735} C_VEL
LIN {X 0,Y 667.201,Z 1018.754,A -85,B 0,C 180,E1 30539.207,E2 30539.207} C_VEL
LIN {X 0,Y 666.626,Z 1041.678,A -85,B 0,C 180,E1 30538.78,E2 30538.78} C_VEL
LIN {X 0,Y 665.892,Z 1063.875,A -85,B 0,C 180,E1 30538.215,E2 30538.215} C_VEL
LIN {X 0,Y 665.041,Z 1086.051,A -85,B 0,C 180,E1 30537.49,E2 30537.49} C_VEL
LIN {X 0,Y 664.018,Z 1107.882,A -85,B 0,C 180,E1 30536.611,E2 30536.611} C_VEL
LIN {X 0,Y 662.952,Z 1129.613,A -85,B 0,C 180,E1 30535.555,E2 30535.555} C_VEL
LIN {X 0,Y 661.815,Z 1150.481,A -85,B 0,C 180,E1 30534.351,E2 30534.351} C_VEL
LIN {X 0,Y 660.756,Z 1170.028,A -85,B 0,C 180,E1 30533.033,E2 30533.033} C_VEL
LIN {X 0,Y 659.7,Z 1189.357,A -85,B 0,C 180,E1 30531.519,E2 30531.519} C_VEL
LIN {X 0,Y 658.779,Z 1206.316,A -85,B 0,C 180,E1 30529.969,E2 30529.969} C_VEL
LIN {X 0,Y 658.078,Z 1220.281,A -85,B 0,C 180,E1 30528.516,E2 30528.516} C_VEL
LIN {X 0,Y 657.482,Z 1233.304,A -85,B 0,C 180,E1 30526.978,E2 30526.978} C_VEL
LIN {X 0,Y 656.951,Z 1246.617,A -85,B 0,C 180,E1 30525.177,E2 30525.177} C_VEL
LIN {X 0,Y 656.519,Z 1258.873,A -85,B 0,C 180,E1 30523.207,E2 30523.207} C_VEL
LIN {X 0,Y 656.261,Z 1268.236,A -85,B 0,C 180,E1 30521.425,E2 30521.425} C_VEL
LIN {X 0,Y 656.094,Z 1276.331,A -85,B 0,C 180,E1 30519.586,E2 30519.586} C_VEL
LIN {X 0,Y 655.98,Z 1284.067,A -85,B 0,C 180,E1 30517.357,E2 30517.357} C_VEL
LIN {X 0,Y 655.919,Z 1288.859,A -85,B 0,C 180,E1 30515.512,E2 30515.512} C_VEL
LIN {X 0,Y 655.899,Z 1292.525,A -85,B 0,C 180,E1 30513.497,E2 30513.497} C_VEL
LIN {X 0,Y 655.897,Z 1294.633,A -85,B 0,C 180,E1 30511.311,E2 30511.311} C_VEL
LIN {X 0,Y 655.894,Z 1294.847,A -85,B 0,C 180,E1 30509.39,E2 30509.39} C_VEL
LIN {X 0,Y 655.898,Z 1293.742,A -85,B 0,C 180,E1 30507.555,E2 30507.555} C_VEL
LIN {X 0,Y 655.906,Z 1291.021,A -85,B 0,C 180,E1 30505.553,E2 30505.553} C_VEL
LIN {X 0,Y 655.937,Z 1286.322,A -85,B 0,C 180,E1 30503.436,E2 30503.436} C_VEL
LIN {X 0,Y 656.021,Z 1280.589,A -85,B 0,C 180,E1 30501.569,E2 30501.569} C_VEL
LIN {X 0,Y 656.128,Z 1273.872,A -85,B 0,C 180,E1 30499.819,E2 30499.819} C_VEL
LIN {X 0,Y 656.345,Z 1265.199,A -85,B 0,C 180,E1 30497.955,E2 30497.955} C_VEL
LIN {X 0,Y 656.701,Z 1253.568,A -85,B 0,C 180,E1 30495.901,E2 30495.901} C_VEL
LIN {X 0,Y 657.075,Z 1242.799,A -85,B 0,C 180,E1 30494.286,E2 30494.286} C_VEL
LIN {X 0,Y 657.591,Z 1230.935,A -85,B 0,C 180,E1 30492.727,E2 30492.727} C_VEL
LIN {X 0,Y 658.294,Z 1216.203,A -85,B 0,C 180,E1 30491.033,E2 30491.033} C_VEL
LIN {X 0,Y 659.174,Z 1198.623,A -85,B 0,C 180,E1 30489.304,E2 30489.304} C_VEL
LIN {X 0,Y 660.005,Z 1183.401,A -85,B 0,C 180,E1 30487.998,E2 30487.998} C_VEL
LIN {X 0,Y 660.995,Z 1165.662,A -85,B 0,C 180,E1 30486.653,E2 30486.653} C_VEL
LIN {X 0,Y 662.082,Z 1145.914,A -85,B 0,C 180,E1 30485.368,E2 30485.368} C_VEL
LIN {X 0,Y 663.162,Z 1125.214,A -85,B 0,C 180,E1 30484.217,E2 30484.217} C_VEL
LIN {X 0,Y 664.256,Z 1103.121,A -85,B 0,C 180,E1 30483.185,E2 30483.185} C_VEL
LIN {X 0,Y 665.232,Z 1080.851,A -85,B 0,C 180,E1 30482.327,E2 30482.327} C_VEL
LIN {X 0,Y 666.101,Z 1057.894,A -85,B 0,C 180,E1 30481.62,E2 30481.62} C_VEL
LIN {X 0,Y 666.818,Z 1035.018,A -85,B 0,C 180,E1 30481.082,E2 30481.082} C_VEL
LIN {X 0,Y 667.314,Z 1011.327,A -85,B 0,C 180,E1 30480.687,E2 30480.687} C_VEL
LIN {X 0,Y 667.757,Z 974.324,A -85,B 0,C 180,E1 30480.241,E2 30480.241} C_VEL
LIN {X 0,Y 672.909,Z 962.507,A -85,B 0,C 180,E1 30479.607,E2 30479.607} C_VEL
LIN {X 0,Y 677.1,Z 955.309,A -85,B 0,C 180,E1 30479.275,E2 30479.275} C_VEL
LIN {X 0,Y 681.947,Z 946.86,A -85,B 0,C 180,E1 30478.902,E2 30478.902} C_VEL
LIN {X 0,Y 688.877,Z 936.901,A -85,B 0,C 180,E1 30478.597,E2 30478.597} C_VEL
LIN {X 0,Y 696.865,Z 925.368,A -85,B 0,C 180,E1 30478.42,E2 30478.42} C_VEL
LIN {X 0,Y 703.499,Z 913.775,A -85,B 0,C 180,E1 30478.361,E2 30478.361} C_VEL
LIN {X 0,Y 706.76,Z 906.507,A -85,B 0,C 180,E1 30478.342,E2 30478.342} C_VEL
LIN {X 0,Y 710.952,Z 895.294,A -85,B 0,C 180,E1 30478.121,E2 30478.121} C_VEL
LIN {X 0,Y 715.29,Z 879.584,A -85,B 0,C 180,E1 30477.939,E2 30477.939} C_VEL
LIN {X 0,Y 717.649,Z 863.835,A -85,B 0,C 180,E1 30477.76,E2 30477.76} C_VEL
LIN {X 0,Y 718.835,Z 851.854,A -85,B 0,C 180,E1 30477.61,E2 30477.61} C_VEL
LIN {X 0,Y 722.528,Z 859.081,A -85,B 0,C 180,E1 30477.102,E2 30477.102} C_VEL
LIN {X 0,Y 723.55,Z 863.32,A -85,B 0,C 180,E1 30476.682,E2 30476.682} C_VEL
LIN {X 0,Y 723.001,Z 866.704,A -85,B 0,C 180,E1 30476.219,E2 30476.219} C_VEL
LIN {X 0,Y 720.878,Z 869.091,A -85,B 0,C 180,E1 30475.729,E2 30475.729} C_VEL
LIN {X 0,Y 717.652,Z 870.151,A -85,B 0,C 180,E1 30475.29,E2 30475.29} C_VEL
LIN {X 0,Y 713.676,Z 869.988,A -85,B 0,C 180,E1 30474.906,E2 30474.906} C_VEL
LIN {X 0,Y 706.173,Z 867.6,A -85,B 0,C 180,E1 30474.365,E2 30474.365} C_VEL
LIN {X 0,Y 696.835,Z 863.04,A -85,B 0,C 180,E1 30473.609,E2 30473.609} C_VEL
LIN {X 0,Y 688.316,Z 856.959,A -85,B 0,C 180,E1 30472.756,E2 30472.756} C_VEL
LIN {X 0,Y 680.797,Z 849.07,A -85,B 0,C 180,E1 30471.791,E2 30471.791} C_VEL
LIN {X 0,Y 674.989,Z 839.781,A -85,B 0,C 180,E1 30470.782,E2 30470.782} C_VEL
LIN {X 0,Y 670.683,Z 828.611,A -85,B 0,C 180,E1 30469.684,E2 30469.684} C_VEL
LIN {X 0,Y 668.242,Z 816.009,A -85,B 0,C 180,E1 30468.56,E2 30468.56} C_VEL
LIN {X 0,Y 667.511,Z 799.655,A -85,B 0,C 180,E1 30467.222,E2 30467.222} C_VEL
LIN {X 0,Y 669.351,Z 758.381,A -85,B 0,C 180,E1 30463.998,E2 30463.998} C_VEL
LIN {X 0,Y 671.046,Z 721.791,A -85,B 0,C 180,E1 30461.068,E2 30461.068} C_VEL
LIN {X 0,Y 672.647,Z 686.993,A -85,B 0,C 180,E1 30458.199,E2 30458.199} C_VEL
LIN {X 0,Y 674.18,Z 653.387,A -85,B 0,C 180,E1 30455.34,E2 30455.34} C_VEL
LIN {X 0,Y 674.325,Z 646.983,A -85,B 0,C 180,E1 30454.771,E2 30454.771} C_VEL
LIN {X 0,Y 665.325,Z 625.908,A -85,B 0,C 180,E1 30451.989,E2 30451.989} C_VEL
LIN {X 0,Y 657.999,Z 609.642,A -85,B 0,C 180,E1 30449.695,E2 30449.695} C_VEL
LIN {X 0,Y 656.7,Z 606.178,A -85,B 0,C 180,E1 30449.196,E2 30449.196} C_VEL
LIN {X 0,Y 656.711,Z 606.178,A -85,B 0,C 180,E1 30446.067,E2 30446.067} C_VEL
LIN {X 0,Y 656.694,Z 606.182,A -85,B 0,C 180,E1 30443.036,E2 30443.036} C_VEL
LIN {X 0,Y 656.706,Z 606.18,A -85,B 0,C 180,E1 30439.942,E2 30439.942} C_VEL
LIN {X 0,Y 656.694,Z 606.177,A -85,B 0,C 180,E1 30436.907,E2 30436.907} C_VEL
LIN {X 0,Y 656.704,Z 606.178,A -85,B 0,C 180,E1 30433.83,E2 30433.83} C_VEL
LIN {X 0,Y 656.696,Z 606.175,A -85,B 0,C 180,E1 30430.705,E2 30430.705} C_VEL
LIN {X 0,Y 656.701,Z 606.177,A -85,B 0,C 180,E1 30427.612,E2 30427.612} C_VEL
LIN {X 0,Y 656.7,Z 606.177,A -85,B 0,C 180,E1 30424.541,E2 30424.541} C_VEL
LIN {X 0,Y 656.7,Z 606.175,A -85,B 0,C 180,E1 30421.396,E2 30421.396} C_VEL
LIN {X 0,Y 656.699,Z 606.175,A -85,B 0,C 180,E1 30418.255,E2 30418.255} C_VEL
LIN {X 0,Y 656.697,Z 606.177,A -85,B 0,C 180,E1 30415.109,E2 30415.109} C_VEL
LIN {X 0,Y 656.701,Z 606.178,A -85,B 0,C 180,E1 30412.036,E2 30412.036} C_VEL
LIN {X 0,Y 656.701,Z 606.178,A -85,B 0,C 180,E1 30408.939,E2 30408.939} C_VEL
LIN {X 0,Y 656.702,Z 606.179,A -85,B 0,C 180,E1 30405.81,E2 30405.81} C_VEL
LIN {X 0,Y 656.698,Z 606.179,A -85,B 0,C 180,E1 30402.637,E2 30402.637} C_VEL
LIN {X 0,Y 656.703,Z 606.18,A -85,B 0,C 180,E1 30399.594,E2 30399.594} C_VEL
LIN {X 0,Y 656.704,Z 606.178,A -85,B 0,C 180,E1 30396.489,E2 30396.489} C_VEL
LIN {X 0,Y 656.705,Z 606.177,A -85,B 0,C 180,E1 30393.407,E2 30393.407} C_VEL
LIN {X 0,Y 656.71,Z 606.181,A -85,B 0,C 180,E1 30390.341,E2 30390.341} C_VEL
LIN {X 0,Y 656.708,Z 606.18,A -85,B 0,C 180,E1 30387.281,E2 30387.281} C_VEL
LIN {X 0,Y 656.703,Z 606.176,A -85,B 0,C 180,E1 30384.22,E2 30384.22} C_VEL
LIN {X 0,Y 656.71,Z 606.175,A -85,B 0,C 180,E1 30381.036,E2 30381.036} C_VEL
LIN {X 0,Y 656.702,Z 606.181,A -85,B 0,C 180,E1 30380.508,E2 30380.508} C_VEL
LIN {X 0,Y 655.708,Z 606.302,A -85,B 0,C 180,E1 30379.836,E2 30379.836} C_VEL
LIN {X 0,Y 649.303,Z 607.099,A -85,B 0,C 180,E1 30377.952,E2 30377.952} C_VEL
LIN {X 0,Y 648.755,Z 607.156,A -85,B 0,C 180,E1 30377.462,E2 30377.462} C_VEL
LIN {X 0,Y 648.771,Z 607.17,A -85,B 0,C 180,E1 30374.347,E2 30374.347} C_VEL
LIN {X 0,Y 648.766,Z 607.159,A -85,B 0,C 180,E1 30371.226,E2 30371.226} C_VEL
LIN {X 0,Y 648.761,Z 607.165,A -85,B 0,C 180,E1 30368.17,E2 30368.17} C_VEL
LIN {X 0,Y 648.772,Z 607.167,A -85,B 0,C 180,E1 30365.077,E2 30365.077} C_VEL
LIN {X 0,Y 648.759,Z 607.173,A -85,B 0,C 180,E1 30361.912,E2 30361.912} C_VEL
LIN {X 0,Y 648.777,Z 607.233,A -85,B 0,C 180,E1 30361.644,E2 30361.644} C_VEL
LIN {X 0,Y 655.356,Z 629.244,A -85,B 0,C 180,E1 30359.926,E2 30359.926} C_VEL
LIN {X 0,Y 654.889,Z 667.067,A -85,B 0,C 180,E1 30357.407,E2 30357.407} C_VEL
LIN {X 0,Y 653.933,Z 710.199,A -85,B 0,C 180,E1 30354.478,E2 30354.478} C_VEL
LIN {X 0,Y 652.874,Z 755.969,A -85,B 0,C 180,E1 30351.375,E2 30351.375} C_VEL
LIN {X 0,Y 651.891,Z 803.217,A -85,B 0,C 180,E1 30348.233,E2 30348.233} C_VEL
LIN {X 0,Y 651.364,Z 834.472,A -85,B 0,C 180,E1 30346.181,E2 30346.181} C_VEL
LIN {X 0,Y 652.192,Z 843.902,A -85,B 0,C 180,E1 30346.051,E2 30346.051} C_VEL
LIN {X 0,Y 651.311,Z 1003.524,A -85,B 0,C 180,E1 30344.249,E2 30344.249} C_VEL
LIN {X 0,Y 651.119,Z 1020.959,A -85,B 0,C 180,E1 30343.89,E2 30343.89} C_VEL
LIN {X 0,Y 650.796,Z 1037.837,A -85,B 0,C 180,E1 30343.368,E2 30343.368} C_VEL
LIN {X 0,Y 650.403,Z 1053.925,A -85,B 0,C 180,E1 30342.698,E2 30342.698} C_VEL
LIN {X 0,Y 649.977,Z 1068.998,A -85,B 0,C 180,E1 30341.895,E2 30341.895} C_VEL
LIN {X 0,Y 649.536,Z 1083.001,A -85,B 0,C 180,E1 30340.958,E2 30340.958} C_VEL
LIN {X 0,Y 649.129,Z 1095.469,A -85,B 0,C 180,E1 30339.933,E2 30339.933} C_VEL
LIN {X 0,Y 648.756,Z 1107.02,A -85,B 0,C 180,E1 30338.775,E2 30338.775} C_VEL
LIN {X 0,Y 648.448,Z 1117.551,A -85,B 0,C 180,E1 30337.477,E2 30337.477} C_VEL
LIN {X 0,Y 648.22,Z 1126.367,A -85,B 0,C 180,E1 30336.108,E2 30336.108} C_VEL
LIN {X 0,Y 648.077,Z 1133.891,A -85,B 0,C 180,E1 30334.6,E2 30334.6} C_VEL
LIN {X 0,Y 647.998,Z 1139.439,A -85,B 0,C 180,E1 30333.095,E2 30333.095} C_VEL
LIN {X 0,Y 647.955,Z 1143.14,A -85,B 0,C 180,E1 30331.59,E2 30331.59} C_VEL
LIN {X 0,Y 647.956,Z 1145.218,A -85,B 0,C 180,E1 30329.999,E2 30329.999} C_VEL
LIN {X 0,Y 647.94,Z 1145.518,A -85,B 0,C 180,E1 30328.407,E2 30328.407} C_VEL
LIN {X 0,Y 647.952,Z 1144,A -85,B 0,C 180,E1 30326.814,E2 30326.814} C_VEL
LIN {X 0,Y 647.977,Z 1140.822,A -85,B 0,C 180,E1 30325.308,E2 30325.308} C_VEL
LIN {X 0,Y 648.049,Z 1135.891,A -85,B 0,C 180,E1 30323.799,E2 30323.799} C_VEL
LIN {X 0,Y 648.168,Z 1129.056,A -85,B 0,C 180,E1 30322.286,E2 30322.286} C_VEL
LIN {X 0,Y 648.365,Z 1120.508,A -85,B 0,C 180,E1 30320.859,E2 30320.859} C_VEL
LIN {X 0,Y 648.651,Z 1110.382,A -85,B 0,C 180,E1 30319.519,E2 30319.519} C_VEL
LIN {X 0,Y 649.001,Z 1099.545,A -85,B 0,C 180,E1 30318.355,E2 30318.355} C_VEL
LIN {X 0,Y 649.403,Z 1087.285,A -85,B 0,C 180,E1 30317.279,E2 30317.279} C_VEL
LIN {X 0,Y 649.841,Z 1073.423,A -85,B 0,C 180,E1 30316.292,E2 30316.292} C_VEL
LIN {X 0,Y 650.279,Z 1058.523,A -85,B 0,C 180,E1 30315.437,E2 30315.437} C_VEL
LIN {X 0,Y 650.693,Z 1042.635,A -85,B 0,C 180,E1 30314.719,E2 30314.719} C_VEL
LIN {X 0,Y 651.034,Z 1025.838,A -85,B 0,C 180,E1 30314.154,E2 30314.154} C_VEL
LIN {X 0,Y 651.279,Z 1007.917,A -85,B 0,C 180,E1 30313.736,E2 30313.736} C_VEL
LIN {X 0,Y 651.414,Z 987.952,A -85,B 0,C 180,E1 30313.465,E2 30313.465} C_VEL
LIN {X 0,Y 651.988,Z 839.545,A -85,B 0,C 180,E1 30311.804,E2 30311.804} C_VEL
LIN {X 0,Y 651.304,Z 833.683,A -85,B 0,C 180,E1 30311.702,E2 30311.702} C_VEL
LIN {X 0,Y 652.233,Z 785.676,A -85,B 0,C 180,E1 30308.521,E2 30308.521} C_VEL
LIN {X 0,Y 653.223,Z 739.815,A -85,B 0,C 180,E1 30305.443,E2 30305.443} C_VEL
LIN {X 0,Y 654.342,Z 694.745,A -85,B 0,C 180,E1 30302.371,E2 30302.371} C_VEL
LIN {X 0,Y 655.19,Z 652.523,A -85,B 0,C 180,E1 30299.506,E2 30299.506} C_VEL
LIN {X 0,Y 655.243,Z 628.144,A -85,B 0,C 180,E1 30297.879,E2 30297.879} C_VEL
LIN {X 0,Y 648.749,Z 607.159,A -85,B 0,C 180,E1 30296.192,E2 30296.192} C_VEL
LIN {X 0,Y 648.765,Z 607.159,A -85,B 0,C 180,E1 30293.163,E2 30293.163} C_VEL
LIN {X 0,Y 648.752,Z 607.153,A -85,B 0,C 180,E1 30290.121,E2 30290.121} C_VEL
LIN {X 0,Y 648.764,Z 607.167,A -85,B 0,C 180,E1 30287.06,E2 30287.06} C_VEL
LIN {X 0,Y 648.758,Z 607.165,A -85,B 0,C 180,E1 30283.913,E2 30283.913} C_VEL
LIN {X 0,Y 648.755,Z 607.166,A -85,B 0,C 180,E1 30280.805,E2 30280.805} C_VEL
LIN {X 0,Y 648.771,Z 607.169,A -85,B 0,C 180,E1 30277.724,E2 30277.724} C_VEL
LIN {X 0,Y 648.757,Z 607.169,A -85,B 0,C 180,E1 30274.554,E2 30274.554} C_VEL
LIN {X 0,Y 648.801,Z 607.402,A -85,B 0,C 180,E1 30271.836,E2 30271.836} C_VEL
LIN {X 0,Y 649.918,Z 610.417,A -85,B 0,C 180,E1 30271.492,E2 30271.492} C_VEL
LIN {X 0,Y 660.554,Z 627.798,A -85,B 0,C 180,E1 30270.579,E2 30270.579} C_VEL
LIN {X 0,Y 663.787,Z 634.052,A -85,B 0,C 180,E1 30270.299,E2 30270.299} C_VEL
LIN {X 0,Y 662.367,Z 737.436,A -85,B 0,C 180,E1 30269.019,E2 30269.019} C_VEL
LIN {X 0,Y 660.387,Z 926.599,A -85,B 0,C 180,E1 30266.766,E2 30266.766} C_VEL
LIN {X 0,Y 659.842,Z 958.101,A -85,B 0,C 180,E1 30266.323,E2 30266.323} C_VEL
LIN {X 0,Y 659.275,Z 978.291,A -85,B 0,C 180,E1 30265.9,E2 30265.9} C_VEL
LIN {X 0,Y 658.627,Z 996.701,A -85,B 0,C 180,E1 30265.404,E2 30265.404} C_VEL
LIN {X 0,Y 657.92,Z 1014.262,A -85,B 0,C 180,E1 30264.827,E2 30264.827} C_VEL
LIN {X 0,Y 657.09,Z 1031.26,A -85,B 0,C 180,E1 30264.163,E2 30264.163} C_VEL
LIN {X 0,Y 656.17,Z 1049.303,A -85,B 0,C 180,E1 30263.341,E2 30263.341} C_VEL
LIN {X 0,Y 654.924,Z 1071.39,A -85,B 0,C 180,E1 30262.154,E2 30262.154} C_VEL
LIN {X 0,Y 653.85,Z 1089.359,A -85,B 0,C 180,E1 30261.015,E2 30261.015} C_VEL
LIN {X 0,Y 652.904,Z 1104.921,A -85,B 0,C 180,E1 30259.895,E2 30259.895} C_VEL
LIN {X 0,Y 652.017,Z 1119.754,A -85,B 0,C 180,E1 30258.694,E2 30258.694} C_VEL
LIN {X 0,Y 651.22,Z 1133.711,A -85,B 0,C 180,E1 30257.422,E2 30257.422} C_VEL
LIN {X 0,Y 650.477,Z 1146.981,A -85,B 0,C 180,E1 30256.063,E2 30256.063} C_VEL
LIN {X 0,Y 649.769,Z 1161.039,A -85,B 0,C 180,E1 30254.436,E2 30254.436} C_VEL
LIN {X 0,Y 649.097,Z 1175.67,A -85,B 0,C 180,E1 30252.454,E2 30252.454} C_VEL
LIN {X 0,Y 648.659,Z 1186.4,A -85,B 0,C 180,E1 30250.75,E2 30250.75} C_VEL
LIN {X 0,Y 648.387,Z 1195.18,A -85,B 0,C 180,E1 30249.14,E2 30249.14} C_VEL
LIN {X 0,Y 648.177,Z 1203.09,A -85,B 0,C 180,E1 30247.445,E2 30247.445} C_VEL
LIN {X 0,Y 648.028,Z 1210.325,A -85,B 0,C 180,E1 30245.578,E2 30245.578} C_VEL
LIN {X 0,Y 647.946,Z 1216.937,A -85,B 0,C 180,E1 30243.362,E2 30243.362} C_VEL
LIN {X 0,Y 647.912,Z 1221.058,A -85,B 0,C 180,E1 30241.415,E2 30241.415} C_VEL
LIN {X 0,Y 647.909,Z 1223.52,A -85,B 0,C 180,E1 30239.646,E2 30239.646} C_VEL
LIN {X 0,Y 647.904,Z 1224.783,A -85,B 0,C 180,E1 30237.789,E2 30237.789} C_VEL
LIN {X 0,Y 647.913,Z 1224.741,A -85,B 0,C 180,E1 30236.018,E2 30236.018} C_VEL
LIN {X 0,Y 647.92,Z 1223.263,A -85,B 0,C 180,E1 30233.976,E2 30233.976} C_VEL
LIN {X 0,Y 647.928,Z 1219.662,A -85,B 0,C 180,E1 30231.748,E2 30231.748} C_VEL
LIN {X 0,Y 647.972,Z 1215.161,A -85,B 0,C 180,E1 30229.902,E2 30229.902} C_VEL
LIN {X 0,Y 648.036,Z 1209.993,A -85,B 0,C 180,E1 30228.248,E2 30228.248} C_VEL
LIN {X 0,Y 648.178,Z 1202.984,A -85,B 0,C 180,E1 30226.439,E2 30226.439} C_VEL
LIN {X 0,Y 648.405,Z 1194.462,A -85,B 0,C 180,E1 30224.619,E2 30224.619} C_VEL
LIN {X 0,Y 648.82,Z 1182.534,A -85,B 0,C 180,E1 30222.512,E2 30222.512} C_VEL
LIN {X 0,Y 649.282,Z 1171.434,A -85,B 0,C 180,E1 30220.851,E2 30220.851} C_VEL
LIN {X 0,Y 649.835,Z 1159.358,A -85,B 0,C 180,E1 30219.274,E2 30219.274} C_VEL
LIN {X 0,Y 650.462,Z 1147.237,A -85,B 0,C 180,E1 30217.876,E2 30217.876} C_VEL
LIN {X 0,Y 651.203,Z 1134.024,A -85,B 0,C 180,E1 30216.519,E2 30216.519} C_VEL
LIN {X 0,Y 652.132,Z 1118.011,A -85,B 0,C 180,E1 30215.061,E2 30215.061} C_VEL
LIN {X 0,Y 653.33,Z 1098.104,A -85,B 0,C 180,E1 30213.504,E2 30213.504} C_VEL
LIN {X 0,Y 654.313,Z 1081.321,A -85,B 0,C 180,E1 30212.368,E2 30212.368} C_VEL
LIN {X 0,Y 655.249,Z 1065.435,A -85,B 0,C 180,E1 30211.419,E2 30211.419} C_VEL
LIN {X 0,Y 656.166,Z 1049.16,A -85,B 0,C 180,E1 30210.565,E2 30210.565} C_VEL
LIN {X 0,Y 657.008,Z 1032.931,A -85,B 0,C 180,E1 30209.819,E2 30209.819} C_VEL
LIN {X 0,Y 657.832,Z 1016.08,A -85,B 0,C 180,E1 30209.149,E2 30209.149} C_VEL
LIN {X 0,Y 658.479,Z 999.966,A -85,B 0,C 180,E1 30208.611,E2 30208.611} C_VEL
LIN {X 0,Y 659.05,Z 981.775,A -85,B 0,C 180,E1 30208.118,E2 30208.118} C_VEL
LIN {X 0,Y 659.522,Z 962.716,A -85,B 0,C 180,E1 30207.713,E2 30207.713} C_VEL
LIN {X 0,Y 659.867,Z 942.891,A -85,B 0,C 180,E1 30207.406,E2 30207.406} C_VEL
LIN {X 0,Y 661.059,Z 696.108,A -85,B 0,C 180,E1 30204.696,E2 30204.696} C_VEL
LIN {X 0,Y 661.246,Z 632.769,A -85,B 0,C 180,E1 30203.98,E2 30203.98} C_VEL
LIN {X 0,Y 657.269,Z 627.046,A -85,B 0,C 180,E1 30203.772,E2 30203.772} C_VEL
LIN {X 0,Y 656.552,Z 626.216,A -85,B 0,C 180,E1 30203.719,E2 30203.719} C_VEL
LIN {X 0,Y 656.373,Z 625.947,A -85,B 0,C 180,E1 30202.674,E2 30202.674} C_VEL
LIN {X 0,Y 657.029,Z 627.341,A -85,B 0,C 180,E1 30201.506,E2 30201.506} C_VEL
LIN {X 0,Y 658.312,Z 630.89,A -85,B 0,C 180,E1 30200.224,E2 30200.224} C_VEL
LIN {X 0,Y 659.375,Z 633.971,A -85,B 0,C 180,E1 30199.483,E2 30199.483} C_VEL
LIN {X 0,Y 655.565,Z 645.016,A -85,B 0,C 180,E1 30198.363,E2 30198.363} C_VEL
LIN {X 0,Y 652.829,Z 657.838,A -85,B 0,C 180,E1 30197.272,E2 30197.272} C_VEL
LIN {X 0,Y 650.86,Z 674.256,A -85,B 0,C 180,E1 30196.097,E2 30196.097} C_VEL
LIN {X 0,Y 649.501,Z 696.824,A -85,B 0,C 180,E1 30194.713,E2 30194.713} C_VEL
LIN {X 0,Y 648.565,Z 734.6,A -85,B 0,C 180,E1 30192.66,E2 30192.66} C_VEL
LIN {X 0,Y 648.805,Z 772.59,A -85,B 0,C 180,E1 30190.686,E2 30190.686} C_VEL
LIN {X 0,Y 650.792,Z 792.867,A -85,B 0,C 180,E1 30189.615,E2 30189.615} C_VEL
LIN {X 0,Y 654.315,Z 809.485,A -85,B 0,C 180,E1 30188.728,E2 30188.728} C_VEL
LIN {X 0,Y 659.393,Z 823.788,A -85,B 0,C 180,E1 30187.952,E2 30187.952} C_VEL
LIN {X 0,Y 665.856,Z 836.558,A -85,B 0,C 180,E1 30187.261,E2 30187.261} C_VEL
LIN {X 0,Y 674.025,Z 848.42,A -85,B 0,C 180,E1 30186.625,E2 30186.625} C_VEL
LIN {X 0,Y 683.087,Z 858.459,A -85,B 0,C 180,E1 30186.098,E2 30186.098} C_VEL
LIN {X 0,Y 693.755,Z 867.705,A -85,B 0,C 180,E1 30185.621,E2 30185.621} C_VEL
LIN {X 0,Y 702.06,Z 873.328,A -85,B 0,C 180,E1 30185.305,E2 30185.305} C_VEL
LIN {X 0,Y 707.084,Z 875.561,A -85,B 0,C 180,E1 30185.038,E2 30185.038} C_VEL
LIN {X 0,Y 712.271,Z 876.661,A -85,B 0,C 180,E1 30184.649,E2 30184.649} C_VEL
LIN {X 0,Y 716.142,Z 876.356,A -85,B 0,C 180,E1 30184.242,E2 30184.242} C_VEL
LIN {X 0,Y 719.199,Z 874.698,A -85,B 0,C 180,E1 30183.758,E2 30183.758} C_VEL
LIN {X 0,Y 720.745,Z 871.87,A -85,B 0,C 180,E1 30183.277,E2 30183.277} C_VEL
LIN {X 0,Y 720.697,Z 868.048,A -85,B 0,C 180,E1 30182.817,E2 30182.817} C_VEL
LIN {X 0,Y 720.597,Z 867.804,A -85,B 0,C 180,E1 30182.781,E2 30182.781} C_VEL
LIN {X 0,Y 716.204,Z 882.754,A -85,B 0,C 180,E1 30182.664,E2 30182.664} C_VEL
LIN {X 0,Y 709.804,Z 897.898,A -85,B 0,C 180,E1 30182.495,E2 30182.495} C_VEL
LIN {X 0,Y 704.967,Z 907.667,A -85,B 0,C 180,E1 30182.291,E2 30182.291} C_VEL
LIN {X 0,Y 697.352,Z 918.867,A -85,B 0,C 180,E1 30182.224,E2 30182.224} C_VEL
LIN {X 0,Y 688.738,Z 929.296,A -85,B 0,C 180,E1 30182.053,E2 30182.053} C_VEL
LIN {X 0,Y 680.357,Z 938.998,A -85,B 0,C 180,E1 30181.746,E2 30181.746} C_VEL
LIN {X 0,Y 673.289,Z 948.409,A -85,B 0,C 180,E1 30181.318,E2 30181.318} C_VEL
LIN {X 0,Y 667.518,Z 957.955,A -85,B 0,C 180,E1 30180.817,E2 30180.817} C_VEL
LIN {X 0,Y 663.258,Z 965.824,A -85,B 0,C 180,E1 30180.384,E2 30180.384} C_VEL
LIN {X 0,Y 660.175,Z 973.57,A -85,B 0,C 180,E1 30179.97,E2 30179.97} C_VEL
LIN {X 0,Y 659.729,Z 1019.055,A -85,B 0,C 180,E1 30179.452,E2 30179.452} C_VEL
LIN {X 0,Y 659.24,Z 1043.65,A -85,B 0,C 180,E1 30179.02,E2 30179.02} C_VEL
LIN {X 0,Y 658.635,Z 1065.856,A -85,B 0,C 180,E1 30178.47,E2 30178.47} C_VEL
LIN {X 0,Y 657.857,Z 1086.485,A -85,B 0,C 180,E1 30177.798,E2 30177.798} C_VEL
LIN {X 0,Y 656.784,Z 1107.803,A -85,B 0,C 180,E1 30176.932,E2 30176.932} C_VEL
LIN {X 0,Y 655.62,Z 1129.527,A -85,B 0,C 180,E1 30175.866,E2 30175.866} C_VEL
LIN {X 0,Y 654.449,Z 1149.553,A -85,B 0,C 180,E1 30174.705,E2 30174.705} C_VEL
LIN {X 0,Y 653.317,Z 1168.644,A -85,B 0,C 180,E1 30173.416,E2 30173.416} C_VEL
LIN {X 0,Y 652.176,Z 1187.46,A -85,B 0,C 180,E1 30171.941,E2 30171.941} C_VEL
LIN {X 0,Y 651.082,Z 1206.215,A -85,B 0,C 180,E1 30170.225,E2 30170.225} C_VEL
LIN {X 0,Y 650.303,Z 1220.273,A -85,B 0,C 180,E1 30168.746,E2 30168.746} C_VEL
LIN {X 0,Y 649.687,Z 1232.572,A -85,B 0,C 180,E1 30167.281,E2 30167.281} C_VEL
LIN {X 0,Y 649.141,Z 1244.292,A -85,B 0,C 180,E1 30165.696,E2 30165.696} C_VEL
LIN {X 0,Y 648.662,Z 1256.835,A -85,B 0,C 180,E1 30163.733,E2 30163.733} C_VEL
LIN {X 0,Y 648.342,Z 1266.938,A -85,B 0,C 180,E1 30161.837,E2 30161.837} C_VEL
LIN {X 0,Y 648.128,Z 1274.961,A -85,B 0,C 180,E1 30160.041,E2 30160.041} C_VEL
LIN {X 0,Y 648.017,Z 1281.544,A -85,B 0,C 180,E1 30158.251,E2 30158.251} C_VEL
LIN {X 0,Y 647.943,Z 1287.671,A -85,B 0,C 180,E1 30156.114,E2 30156.114} C_VEL
LIN {X 0,Y 647.915,Z 1291.576,A -85,B 0,C 180,E1 30154.161,E2 30154.161} C_VEL
LIN {X 0,Y 647.904,Z 1293.98,A -85,B 0,C 180,E1 30152.212,E2 30152.212} C_VEL
LIN {X 0,Y 647.898,Z 1294.939,A -85,B 0,C 180,E1 30150.266,E2 30150.266} C_VEL
LIN {X 0,Y 647.906,Z 1294.225,A -85,B 0,C 180,E1 30148.056,E2 30148.056} C_VEL
LIN {X 0,Y 647.906,Z 1291.983,A -85,B 0,C 180,E1 30146.108,E2 30146.108} C_VEL
LIN {X 0,Y 647.92,Z 1288.462,A -85,B 0,C 180,E1 30144.244,E2 30144.244} C_VEL
LIN {X 0,Y 647.979,Z 1283.291,A -85,B 0,C 180,E1 30142.286,E2 30142.286} C_VEL
LIN {X 0,Y 648.116,Z 1275.728,A -85,B 0,C 180,E1 30140.141,E2 30140.141} C_VEL
LIN {X 0,Y 648.329,Z 1267.376,A -85,B 0,C 180,E1 30138.255,E2 30138.255} C_VEL
LIN {X 0,Y 648.621,Z 1257.858,A -85,B 0,C 180,E1 30136.45,E2 30136.45} C_VEL
LIN {X 0,Y 649.129,Z 1244.737,A -85,B 0,C 180,E1 30134.363,E2 30134.363} C_VEL
LIN {X 0,Y 649.687,Z 1232.602,A -85,B 0,C 180,E1 30132.722,E2 30132.722} C_VEL
LIN {X 0,Y 650.346,Z 1219.478,A -85,B 0,C 180,E1 30131.165,E2 30131.165} C_VEL
LIN {X 0,Y 651.192,Z 1204.499,A -85,B 0,C 180,E1 30129.603,E2 30129.603} C_VEL
LIN {X 0,Y 652.259,Z 1186.025,A -85,B 0,C 180,E1 30127.942,E2 30127.942} C_VEL
LIN {X 0,Y 653.381,Z 1167.63,A -85,B 0,C 180,E1 30126.508,E2 30126.508} C_VEL
LIN {X 0,Y 654.59,Z 1147.468,A -85,B 0,C 180,E1 30125.163,E2 30125.163} C_VEL
LIN {X 0,Y 655.756,Z 1127.036,A -85,B 0,C 180,E1 30124.001,E2 30124.001} C_VEL
LIN {X 0,Y 656.897,Z 1105.737,A -85,B 0,C 180,E1 30122.978,E2 30122.978} C_VEL
LIN {X 0,Y 657.944,Z 1084.458,A -85,B 0,C 180,E1 30122.129,E2 30122.129} C_VEL
LIN {X 0,Y 658.811,Z 1061.769,A -85,B 0,C 180,E1 30121.404,E2 30121.404} C_VEL
LIN {X 0,Y 659.669,Z 1037.437,A -85,B 0,C 180,E1 30120.805,E2 30120.805} C_VEL
LIN {X 0,Y 660.263,Z 1013.938,A -85,B 0,C 180,E1 30120.387,E2 30120.387} C_VEL
LIN {X 0,Y 660.934,Z 972.823,A -85,B 0,C 180,E1 30119.877,E2 30119.877} C_VEL
LIN {X 0,Y 666.451,Z 960.713,A -85,B 0,C 180,E1 30119.231,E2 30119.231} C_VEL
LIN {X 0,Y 670.61,Z 953.661,A -85,B 0,C 180,E1 30118.895,E2 30118.895} C_VEL
LIN {X 0,Y 676.066,Z 944.709,A -85,B 0,C 180,E1 30118.48,E2 30118.48} C_VEL
LIN {X 0,Y 683.986,Z 934.735,A -85,B 0,C 180,E1 30118.1,E2 30118.1} C_VEL
LIN {X 0,Y 693.191,Z 924.077,A -85,B 0,C 180,E1 30117.843,E2 30117.843} C_VEL
LIN {X 0,Y 701.702,Z 912.818,A -85,B 0,C 180,E1 30117.73,E2 30117.73} C_VEL
LIN {X 0,Y 705.313,Z 907.006,A -85,B 0,C 180,E1 30117.695,E2 30117.695} C_VEL
LIN {X 0,Y 710.81,Z 895.764,A -85,B 0,C 180,E1 30117.474,E2 30117.474} C_VEL
LIN {X 0,Y 716.703,Z 881.345,A -85,B 0,C 180,E1 30117.324,E2 30117.324} C_VEL
LIN {X 0,Y 720.647,Z 867.816,A -85,B 0,C 180,E1 30117.206,E2 30117.206} C_VEL
LIN {X 0,Y 720.812,Z 871.541,A -85,B 0,C 180,E1 30116.769,E2 30116.769} C_VEL
LIN {X 0,Y 719.599,Z 874.258,A -85,B 0,C 180,E1 30116.331,E2 30116.331} C_VEL
LIN {X 0,Y 717.23,Z 875.983,A -85,B 0,C 180,E1 30115.904,E2 30115.904} C_VEL
LIN {X 0,Y 713.609,Z 876.697,A -85,B 0,C 180,E1 30115.477,E2 30115.477} C_VEL
LIN {X 0,Y 708.637,Z 876.031,A -85,B 0,C 180,E1 30115.065,E2 30115.065} C_VEL
LIN {X 0,Y 697.316,Z 871.779,A -85,B 0,C 180,E1 30114.252,E2 30114.252} C_VEL
LIN {X 0,Y 687.583,Z 866.207,A -85,B 0,C 180,E1 30113.391,E2 30113.391} C_VEL
LIN {X 0,Y 679.407,Z 859.468,A -85,B 0,C 180,E1 30112.491,E2 30112.491} C_VEL
LIN {X 0,Y 672.763,Z 851.648,A -85,B 0,C 180,E1 30111.56,E2 30111.56} C_VEL
LIN {X 0,Y 667.229,Z 841.893,A -85,B 0,C 180,E1 30110.513,E2 30110.513} C_VEL
LIN {X 0,Y 663.341,Z 830.935,A -85,B 0,C 180,E1 30109.439,E2 30109.439} C_VEL
LIN {X 0,Y 661.054,Z 817.976,A -85,B 0,C 180,E1 30108.279,E2 30108.279} C_VEL
LIN {X 0,Y 660.495,Z 800.657,A -85,B 0,C 180,E1 30106.86,E2 30106.86} C_VEL
LIN {X 0,Y 662.446,Z 760.534,A -85,B 0,C 180,E1 30103.7,E2 30103.7} C_VEL
LIN {X 0,Y 664.3,Z 723.804,A -85,B 0,C 180,E1 30100.73,E2 30100.73} C_VEL
LIN {X 0,Y 666.021,Z 689.12,A -85,B 0,C 180,E1 30097.848,E2 30097.848} C_VEL
LIN {X 0,Y 667.668,Z 655.369,A -85,B 0,C 180,E1 30094.953,E2 30094.953} C_VEL
LIN {X 0,Y 667.732,Z 651.012,A -85,B 0,C 180,E1 30094.557,E2 30094.557} C_VEL
LIN {X 0,Y 658.818,Z 630.203,A -85,B 0,C 180,E1 30091.779,E2 30091.779} C_VEL
LIN {X 0,Y 651.644,Z 614.239,A -85,B 0,C 180,E1 30089.508,E2 30089.508} C_VEL
LIN {X 0,Y 649.637,Z 609.908,A -85,B 0,C 180,E1 30088.867,E2 30088.867} C_VEL
LIN {X 0,Y 648.767,Z 607.17,A -85,B 0,C 180,E1 30088.478,E2 30088.478} C_VEL
LIN {X 0,Y 648.764,Z 607.17,A -85,B 0,C 180,E1 30085.37,E2 30085.37} C_VEL
LIN {X 0,Y 648.761,Z 607.169,A -85,B 0,C 180,E1 30082.185,E2 30082.185} C_VEL
LIN {X 0,Y 648.76,Z 607.166,A -85,B 0,C 180,E1 30079.071,E2 30079.071} C_VEL
LIN {X 0,Y 648.759,Z 607.168,A -85,B 0,C 180,E1 30075.91,E2 30075.91} C_VEL
LIN {X 0,Y 648.76,Z 607.167,A -85,B 0,C 180,E1 30072.823,E2 30072.823} C_VEL
LIN {X 0,Y 648.758,Z 607.169,A -85,B 0,C 180,E1 30069.671,E2 30069.671} C_VEL
LIN {X 0,Y 648.765,Z 607.165,A -85,B 0,C 180,E1 30066.638,E2 30066.638} C_VEL
LIN {X 0,Y 648.763,Z 607.167,A -85,B 0,C 180,E1 30063.534,E2 30063.534} C_VEL
LIN {X 0,Y 648.77,Z 607.168,A -85,B 0,C 180,E1 30060.442,E2 30060.442} C_VEL
LIN {X 0,Y 648.767,Z 607.17,A -85,B 0,C 180,E1 30057.35,E2 30057.35} C_VEL
LIN {X 0,Y 648.769,Z 607.17,A -85,B 0,C 180,E1 30054.25,E2 30054.25} C_VEL
LIN {X 0,Y 648.77,Z 607.17,A -85,B 0,C 180,E1 30051.134,E2 30051.134} C_VEL
LIN {X 0,Y 648.77,Z 607.169,A -85,B 0,C 180,E1 30047.991,E2 30047.991} C_VEL
LIN {X 0,Y 648.777,Z 607.169,A -85,B 0,C 180,E1 30044.811,E2 30044.811} C_VEL
LIN {X 0,Y 648.769,Z 607.169,A -85,B 0,C 180,E1 30041.675,E2 30041.675} C_VEL
LIN {X 0,Y 648.776,Z 607.168,A -85,B 0,C 180,E1 30038.481,E2 30038.481} C_VEL
LIN {X 0,Y 648.764,Z 607.167,A -85,B 0,C 180,E1 30035.312,E2 30035.312} C_VEL
LIN {X 0,Y 648.773,Z 607.163,A -85,B 0,C 180,E1 30032.161,E2 30032.161} C_VEL
LIN {X 0,Y 648.758,Z 607.166,A -85,B 0,C 180,E1 30029.017,E2 30029.017} C_VEL
LIN {X 0,Y 648.768,Z 607.167,A -85,B 0,C 180,E1 30025.875,E2 30025.875} C_VEL
LIN {X 0,Y 648.758,Z 607.168,A -85,B 0,C 180,E1 30022.824,E2 30022.824} C_VEL
LIN {X 0,Y 648.765,Z 607.167,A -85,B 0,C 180,E1 30019.718,E2 30019.718} C_VEL
LIN {X 0,Y 648.755,Z 607.156,A -85,B 0,C 180,E1 30017.462,E2 30017.462} C_VEL
LIN {X 0,Y 647.749,Z 607.277,A -85,B 0,C 180,E1 30016.782,E2 30016.782} C_VEL
LIN {X 0,Y 641.359,Z 608.086,A -85,B 0,C 180,E1 30014.874,E2 30014.874} C_VEL
LIN {X 0,Y 640.832,Z 608.158,A -85,B 0,C 180,E1 30014.378,E2 30014.378} C_VEL
LIN {X 0,Y 640.827,Z 608.146,A -85,B 0,C 180,E1 30011.23,E2 30011.23} C_VEL
LIN {X 0,Y 640.824,Z 608.153,A -85,B 0,C 180,E1 30008.149,E2 30008.149} C_VEL
LIN {X 0,Y 640.832,Z 608.154,A -85,B 0,C 180,E1 30004.999,E2 30004.999} C_VEL
LIN {X 0,Y 640.824,Z 608.192,A -85,B 0,C 180,E1 30001.946,E2 30001.946} C_VEL
LIN {X 0,Y 647.926,Z 631.556,A -85,B 0,C 180,E1 30000.1,E2 30000.1} C_VEL
LIN {X 0,Y 647.421,Z 668.115,A -85,B 0,C 180,E1 29997.65,E2 29997.65} C_VEL
LIN {X 0,Y 646.433,Z 710.262,A -85,B 0,C 180,E1 29994.774,E2 29994.774} C_VEL
LIN {X 0,Y 645.316,Z 755.207,A -85,B 0,C 180,E1 29991.702,E2 29991.702} C_VEL
LIN {X 0,Y 644.273,Z 802.874,A -85,B 0,C 180,E1 29988.512,E2 29988.512} C_VEL
LIN {X 0,Y 643.75,Z 835.348,A -85,B 0,C 180,E1 29986.391,E2 29986.391} C_VEL
LIN {X 0,Y 644.572,Z 844.654,A -85,B 0,C 180,E1 29986.26,E2 29986.26} C_VEL
LIN {X 0,Y 643.624,Z 1004.488,A -85,B 0,C 180,E1 29984.434,E2 29984.434} C_VEL
LIN {X 0,Y 643.429,Z 1021.92,A -85,B 0,C 180,E1 29984.071,E2 29984.071} C_VEL
LIN {X 0,Y 643.121,Z 1037.887,A -85,B 0,C 180,E1 29983.576,E2 29983.576} C_VEL
LIN {X 0,Y 642.705,Z 1054.168,A -85,B 0,C 180,E1 29982.899,E2 29982.899} C_VEL
LIN {X 0,Y 642.251,Z 1069.377,A -85,B 0,C 180,E1 29982.086,E2 29982.086} C_VEL
LIN {X 0,Y 641.782,Z 1083.524,A -85,B 0,C 180,E1 29981.138,E2 29981.138} C_VEL
LIN {X 0,Y 641.323,Z 1096.551,A -85,B 0,C 180,E1 29980.055,E2 29980.055} C_VEL
LIN {X 0,Y 640.92,Z 1108.082,A -85,B 0,C 180,E1 29978.883,E2 29978.883} C_VEL
LIN {X 0,Y 640.593,Z 1118.209,A -85,B 0,C 180,E1 29977.622,E2 29977.622} C_VEL
LIN {X 0,Y 640.344,Z 1126.894,A -85,B 0,C 180,E1 29976.274,E2 29976.274} C_VEL
LIN {X 0,Y 640.172,Z 1134.311,A -85,B 0,C 180,E1 29974.793,E2 29974.793} C_VEL
LIN {X 0,Y 640.075,Z 1140.142,A -85,B 0,C 180,E1 29973.223,E2 29973.223} C_VEL
LIN {X 0,Y 640.019,Z 1143.96,A -85,B 0,C 180,E1 29971.7,E2 29971.7} C_VEL
LIN {X 0,Y 640.012,Z 1146.115,A -85,B 0,C 180,E1 29970.088,E2 29970.088} C_VEL
LIN {X 0,Y 639.997,Z 1146.489,A -85,B 0,C 180,E1 29968.477,E2 29968.477} C_VEL
LIN {X 0,Y 640.013,Z 1145.079,A -85,B 0,C 180,E1 29966.864,E2 29966.864} C_VEL
LIN {X 0,Y 640.045,Z 1141.984,A -85,B 0,C 180,E1 29965.339,E2 29965.339} C_VEL
LIN {X 0,Y 640.132,Z 1136.796,A -85,B 0,C 180,E1 29963.722,E2 29963.722} C_VEL
LIN {X 0,Y 640.273,Z 1129.942,A -85,B 0,C 180,E1 29962.19,E2 29962.19} C_VEL
LIN {X 0,Y 640.496,Z 1121.372,A -85,B 0,C 180,E1 29960.746,E2 29960.746} C_VEL
LIN {X 0,Y 640.814,Z 1111.225,A -85,B 0,C 180,E1 29959.389,E2 29959.389} C_VEL
LIN {X 0,Y 641.197,Z 1100.364,A -85,B 0,C 180,E1 29958.211,E2 29958.211} C_VEL
LIN {X 0,Y 641.629,Z 1088.059,A -85,B 0,C 180,E1 29957.123,E2 29957.123} C_VEL
LIN {X 0,Y 642.099,Z 1074.158,A -85,B 0,C 180,E1 29956.124,E2 29956.124} C_VEL
LIN {X 0,Y 642.571,Z 1059.019,A -85,B 0,C 180,E1 29955.248,E2 29955.248} C_VEL
LIN {X 0,Y 642.999,Z 1043.218,A -85,B 0,C 180,E1 29954.532,E2 29954.532} C_VEL
LIN {X 0,Y 643.352,Z 1026.222,A -85,B 0,C 180,E1 29953.959,E2 29953.959} C_VEL
LIN {X 0,Y 643.596,Z 1008.544,A -85,B 0,C 180,E1 29953.545,E2 29953.545} C_VEL
LIN {X 0,Y 643.732,Z 987.95,A -85,B 0,C 180,E1 29953.266,E2 29953.266} C_VEL
LIN {X 0,Y 644.369,Z 840.321,A -85,B 0,C 180,E1 29951.594,E2 29951.594} C_VEL
LIN {X 0,Y 643.701,Z 834.765,A -85,B 0,C 180,E1 29951.501,E2 29951.501} C_VEL
LIN {X 0,Y 644.646,Z 784.813,A -85,B 0,C 180,E1 29948.199,E2 29948.199} C_VEL
LIN {X 0,Y 645.721,Z 738.886,A -85,B 0,C 180,E1 29945.089,E2 29945.089} C_VEL
LIN {X 0,Y 646.878,Z 694.948,A -85,B 0,C 180,E1 29942.072,E2 29942.072} C_VEL
LIN {X 0,Y 647.782,Z 653.184,A -85,B 0,C 180,E1 29939.223,E2 29939.223} C_VEL
LIN {X 0,Y 647.881,Z 630.839,A -85,B 0,C 180,E1 29937.724,E2 29937.724} C_VEL
LIN {X 0,Y 640.819,Z 608.148,A -85,B 0,C 180,E1 29935.878,E2 29935.878} C_VEL
LIN {X 0,Y 640.832,Z 608.152,A -85,B 0,C 180,E1 29932.727,E2 29932.727} C_VEL
LIN {X 0,Y 640.821,Z 608.142,A -85,B 0,C 180,E1 29929.592,E2 29929.592} C_VEL
LIN {X 0,Y 640.828,Z 608.152,A -85,B 0,C 180,E1 29926.385,E2 29926.385} C_VEL
LIN {X 0,Y 640.827,Z 608.157,A -85,B 0,C 180,E1 29923.112,E2 29923.112} C_VEL
LIN {X 0,Y 640.835,Z 608.153,A -85,B 0,C 180,E1 29919.994,E2 29919.994} C_VEL
LIN {X 0,Y 640.825,Z 608.156,A -85,B 0,C 180,E1 29916.81,E2 29916.81} C_VEL
LIN {X 0,Y 640.835,Z 608.161,A -85,B 0,C 180,E1 29913.635,E2 29913.635} C_VEL
LIN {X 0,Y 640.83,Z 608.268,A -85,B 0,C 180,E1 29912.421,E2 29912.421} C_VEL
LIN {X 0,Y 642.328,Z 611.968,A -85,B 0,C 180,E1 29911.963,E2 29911.963} C_VEL
LIN {X 0,Y 655.056,Z 632.746,A -85,B 0,C 180,E1 29910.847,E2 29910.847} C_VEL
LIN {X 0,Y 657.148,Z 636.914,A -85,B 0,C 180,E1 29910.658,E2 29910.658} C_VEL
LIN {X 0,Y 654.92,Z 791.924,A -85,B 0,C 180,E1 29908.729,E2 29908.729} C_VEL
LIN {X 0,Y 653.546,Z 903.737,A -85,B 0,C 180,E1 29907.363,E2 29907.363} C_VEL
LIN {X 0,Y 652.912,Z 952.084,A -85,B 0,C 180,E1 29906.75,E2 29906.75} C_VEL
LIN {X 0,Y 652.197,Z 976.752,A -85,B 0,C 180,E1 29906.262,E2 29906.262} C_VEL
LIN {X 0,Y 651.445,Z 997.175,A -85,B 0,C 180,E1 29905.713,E2 29905.713} C_VEL
LIN {X 0,Y 650.658,Z 1015.659,A -85,B 0,C 180,E1 29905.096,E2 29905.096} C_VEL
LIN {X 0,Y 649.559,Z 1037.522,A -85,B 0,C 180,E1 29904.22,E2 29904.22} C_VEL
LIN {X 0,Y 648.307,Z 1058.947,A -85,B 0,C 180,E1 29903.159,E2 29903.159} C_VEL
LIN {X 0,Y 647.314,Z 1075.008,A -85,B 0,C 180,E1 29902.238,E2 29902.238} C_VEL
LIN {X 0,Y 646.311,Z 1090.59,A -85,B 0,C 180,E1 29901.224,E2 29901.224} C_VEL
LIN {X 0,Y 645.362,Z 1105.082,A -85,B 0,C 180,E1 29900.165,E2 29900.165} C_VEL
LIN {X 0,Y 644.442,Z 1119.149,A -85,B 0,C 180,E1 29899.016,E2 29899.016} C_VEL
LIN {X 0,Y 643.568,Z 1133.17,A -85,B 0,C 180,E1 29897.729,E2 29897.729} C_VEL
LIN {X 0,Y 642.812,Z 1145.656,A -85,B 0,C 180,E1 29896.445,E2 29896.445} C_VEL
LIN {X 0,Y 642.124,Z 1157.598,A -85,B 0,C 180,E1 29895.073,E2 29895.073} C_VEL
LIN {X 0,Y 641.506,Z 1169.57,A -85,B 0,C 180,E1 29893.521,E2 29893.521} C_VEL
LIN {X 0,Y 640.946,Z 1181.817,A -85,B 0,C 180,E1 29891.701,E2 29891.701} C_VEL
LIN {X 0,Y 640.484,Z 1193.571,A -85,B 0,C 180,E1 29889.616,E2 29889.616} C_VEL
LIN {X 0,Y 640.235,Z 1201.71,A -85,B 0,C 180,E1 29887.899,E2 29887.899} C_VEL
LIN {X 0,Y 640.071,Z 1208.845,A -85,B 0,C 180,E1 29886.098,E2 29886.098} C_VEL
LIN {X 0,Y 639.987,Z 1214.344,A -85,B 0,C 180,E1 29884.391,E2 29884.391} C_VEL
LIN {X 0,Y 639.939,Z 1218.854,A -85,B 0,C 180,E1 29882.597,E2 29882.597} C_VEL
LIN {X 0,Y 639.922,Z 1222.669,A -85,B 0,C 180,E1 29880.448,E2 29880.448} C_VEL
LIN {X 0,Y 639.914,Z 1224.598,A -85,B 0,C 180,E1 29878.299,E2 29878.299} C_VEL
LIN {X 0,Y 639.913,Z 1224.848,A -85,B 0,C 180,E1 29876.417,E2 29876.417} C_VEL
LIN {X 0,Y 639.911,Z 1223.964,A -85,B 0,C 180,E1 29874.71,E2 29874.71} C_VEL
LIN {X 0,Y 639.922,Z 1221.675,A -85,B 0,C 180,E1 29872.819,E2 29872.819} C_VEL
LIN {X 0,Y 639.943,Z 1218.001,A -85,B 0,C 180,E1 29870.92,E2 29870.92} C_VEL
LIN {X 0,Y 640.024,Z 1211.738,A -85,B 0,C 180,E1 29868.647,E2 29868.647} C_VEL
LIN {X 0,Y 640.171,Z 1204.511,A -85,B 0,C 180,E1 29866.675,E2 29866.675} C_VEL
LIN {X 0,Y 640.38,Z 1196.51,A -85,B 0,C 180,E1 29864.885,E2 29864.885} C_VEL
LIN {X 0,Y 640.677,Z 1188.247,A -85,B 0,C 180,E1 29863.312,E2 29863.312} C_VEL
LIN {X 0,Y 641.071,Z 1178.708,A -85,B 0,C 180,E1 29861.729,E2 29861.729} C_VEL
LIN {X 0,Y 641.663,Z 1166.403,A -85,B 0,C 180,E1 29859.951,E2 29859.951} C_VEL
LIN {X 0,Y 642.51,Z 1150.983,A -85,B 0,C 180,E1 29858.051,E2 29858.051} C_VEL
LIN {X 0,Y 643.335,Z 1136.958,A -85,B 0,C 180,E1 29856.554,E2 29856.554} C_VEL
LIN {X 0,Y 644.216,Z 1122.906,A -85,B 0,C 180,E1 29855.224,E2 29855.224} C_VEL
LIN {X 0,Y 645.156,Z 1108.165,A -85,B 0,C 180,E1 29853.985,E2 29853.985} C_VEL
LIN {X 0,Y 646.119,Z 1093.472,A -85,B 0,C 180,E1 29852.887,E2 29852.887} C_VEL
LIN {X 0,Y 647.136,Z 1077.785,A -85,B 0,C 180,E1 29851.844,E2 29851.844} C_VEL
LIN {X 0,Y 648.174,Z 1061.252,A -85,B 0,C 180,E1 29850.876,E2 29850.876} C_VEL
LIN {X 0,Y 649.074,Z 1045.057,A -85,B 0,C 180,E1 29850.058,E2 29850.058} C_VEL
LIN {X 0,Y 650.118,Z 1023.586,A -85,B 0,C 180,E1 29849.141,E2 29849.141} C_VEL
LIN {X 0,Y 650.962,Z 1002.167,A -85,B 0,C 180,E1 29848.414,E2 29848.414} C_VEL
LIN {X 0,Y 651.578,Z 982.401,A -85,B 0,C 180,E1 29847.874,E2 29847.874} C_VEL
LIN {X 0,Y 652.094,Z 959.837,A -85,B 0,C 180,E1 29847.409,E2 29847.409} C_VEL
LIN {X 0,Y 652.485,Z 930.583,A -85,B 0,C 180,E1 29847.021,E2 29847.021} C_VEL
LIN {X 0,Y 653.686,Z 681.604,A -85,B 0,C 180,E1 29844.279,E2 29844.279} C_VEL
LIN {X 0,Y 653.817,Z 635.418,A -85,B 0,C 180,E1 29843.743,E2 29843.743} C_VEL
LIN {X 0,Y 651.01,Z 631.927,A -85,B 0,C 180,E1 29843.593,E2 29843.593} C_VEL
LIN {X 0,Y 650.16,Z 630.974,A -85,B 0,C 180,E1 29843.546,E2 29843.546} C_VEL
LIN {X 0,Y 650.129,Z 630.996,A -85,B 0,C 180,E1 29842.479,E2 29842.479} C_VEL
LIN {X 0,Y 650.749,Z 632.438,A -85,B 0,C 180,E1 29841.453,E2 29841.453} C_VEL
LIN {X 0,Y 652.02,Z 635.989,A -85,B 0,C 180,E1 29840.202,E2 29840.202} C_VEL
LIN {X 0,Y 652.661,Z 637.932,A -85,B 0,C 180,E1 29839.721,E2 29839.721} C_VEL
LIN {X 0,Y 648.481,Z 649.176,A -85,B 0,C 180,E1 29838.536,E2 29838.536} C_VEL
LIN {X 0,Y 645.454,Z 662.273,A -85,B 0,C 180,E1 29837.379,E2 29837.379} C_VEL
LIN {X 0,Y 643.371,Z 677.878,A -85,B 0,C 180,E1 29836.212,E2 29836.212} C_VEL
LIN {X 0,Y 641.856,Z 699.404,A -85,B 0,C 180,E1 29834.831,E2 29834.831} C_VEL
LIN {X 0,Y 640.801,Z 733.188,A -85,B 0,C 180,E1 29832.917,E2 29832.917} C_VEL
LIN {X 0,Y 640.885,Z 773.171,A -85,B 0,C 180,E1 29830.778,E2 29830.778} C_VEL
LIN {X 0,Y 642.716,Z 792.866,A -85,B 0,C 180,E1 29829.715,E2 29829.715} C_VEL
LIN {X 0,Y 645.958,Z 809.204,A -85,B 0,C 180,E1 29828.823,E2 29828.823} C_VEL
LIN {X 0,Y 650.928,Z 824.119,A -85,B 0,C 180,E1 29827.999,E2 29827.999} C_VEL
LIN {X 0,Y 657.464,Z 837.678,A -85,B 0,C 180,E1 29827.251,E2 29827.251} C_VEL
LIN {X 0,Y 665.517,Z 849.944,A -85,B 0,C 180,E1 29826.578,E2 29826.578} C_VEL
LIN {X 0,Y 674.784,Z 860.718,A -85,B 0,C 180,E1 29825.995,E2 29825.995} C_VEL
LIN {X 0,Y 685.725,Z 870.704,A -85,B 0,C 180,E1 29825.475,E2 29825.475} C_VEL
LIN {X 0,Y 697.349,Z 878.939,A -85,B 0,C 180,E1 29825.042,E2 29825.042} C_VEL
LIN {X 0,Y 702.623,Z 881.538,A -85,B 0,C 180,E1 29824.803,E2 29824.803} C_VEL
LIN {X 0,Y 708.071,Z 882.999,A -85,B 0,C 180,E1 29824.443,E2 29824.443} C_VEL
LIN {X 0,Y 712.149,Z 883.048,A -85,B 0,C 180,E1 29824.066,E2 29824.066} C_VEL
LIN {X 0,Y 715.707,Z 881.759,A -85,B 0,C 180,E1 29823.59,E2 29823.59} C_VEL
LIN {X 0,Y 716.925,Z 880.746,A -85,B 0,C 180,E1 29823.323,E2 29823.323} C_VEL
LIN {X 0,Y 709.228,Z 894.854,A -85,B 0,C 180,E1 29823.163,E2 29823.163} C_VEL
LIN {X 0,Y 702.336,Z 906.044,A -85,B 0,C 180,E1 29822.919,E2 29822.919} C_VEL
LIN {X 0,Y 697.332,Z 912.244,A -85,B 0,C 180,E1 29822.833,E2 29822.833} C_VEL
LIN {X 0,Y 687.952,Z 921.952,A -85,B 0,C 180,E1 29822.632,E2 29822.632} C_VEL
LIN {X 0,Y 678.064,Z 931.544,A -85,B 0,C 180,E1 29822.264,E2 29822.264} C_VEL
LIN {X 0,Y 669.521,Z 940.94,A -85,B 0,C 180,E1 29821.766,E2 29821.766} C_VEL
LIN {X 0,Y 663.572,Z 949.763,A -85,B 0,C 180,E1 29821.273,E2 29821.273} C_VEL
LIN {X 0,Y 656.412,Z 961.908,A -85,B 0,C 180,E1 29820.583,E2 29820.583} C_VEL
LIN {X 0,Y 653.386,Z 968.875,A -85,B 0,C 180,E1 29820.209,E2 29820.209} C_VEL
LIN {X 0,Y 652.426,Z 975.761,A -85,B 0,C 180,E1 29820.159,E2 29820.159} C_VEL
LIN {X 0,Y 652.07,Z 1015.786,A -85,B 0,C 180,E1 29819.687,E2 29819.687} C_VEL
LIN {X 0,Y 651.516,Z 1041.725,A -85,B 0,C 180,E1 29819.222,E2 29819.222} C_VEL
LIN {X 0,Y 650.825,Z 1067.006,A -85,B 0,C 180,E1 29818.606,E2 29818.606} C_VEL
LIN {X 0,Y 650.04,Z 1091.119,A -85,B 0,C 180,E1 29817.855,E2 29817.855} C_VEL
LIN {X 0,Y 649.239,Z 1111.04,A -85,B 0,C 180,E1 29817.077,E2 29817.077} C_VEL
LIN {X 0,Y 648.297,Z 1129.6,A -85,B 0,C 180,E1 29816.175,E2 29816.175} C_VEL
LIN {X 0,Y 647.043,Z 1149.621,A -85,B 0,C 180,E1 29815.003,E2 29815.003} C_VEL
LIN {X 0,Y 645.797,Z 1168.833,A -85,B 0,C 180,E1 29813.691,E2 29813.691} C_VEL
LIN {X 0,Y 644.603,Z 1187.118,A -85,B 0,C 180,E1 29812.241,E2 29812.241} C_VEL
LIN {X 0,Y 643.447,Z 1205.391,A -85,B 0,C 180,E1 29810.561,E2 29810.561} C_VEL
LIN {X 0,Y 642.589,Z 1219.451,A -85,B 0,C 180,E1 29809.074,E2 29809.074} C_VEL
LIN {X 0,Y 641.894,Z 1231.97,A -85,B 0,C 180,E1 29807.574,E2 29807.574} C_VEL
LIN {X 0,Y 641.337,Z 1242.758,A -85,B 0,C 180,E1 29806.113,E2 29806.113} C_VEL
LIN {X 0,Y 640.891,Z 1252.961,A -85,B 0,C 180,E1 29804.549,E2 29804.549} C_VEL
LIN {X 0,Y 640.484,Z 1263.815,A -85,B 0,C 180,E1 29802.626,E2 29802.626} C_VEL
LIN {X 0,Y 640.199,Z 1273.489,A -85,B 0,C 180,E1 29800.53,E2 29800.53} C_VEL
LIN {X 0,Y 640.04,Z 1280.012,A -85,B 0,C 180,E1 29798.808,E2 29798.808} C_VEL
LIN {X 0,Y 639.964,Z 1285.308,A -85,B 0,C 180,E1 29797.091,E2 29797.091} C_VEL
LIN {X 0,Y 639.929,Z 1289.802,A -85,B 0,C 180,E1 29795.201,E2 29795.201} C_VEL
LIN {X 0,Y 639.907,Z 1293.331,A -85,B 0,C 180,E1 29792.957,E2 29792.957} C_VEL
LIN {X 0,Y 639.906,Z 1294.761,A -85,B 0,C 180,E1 29790.897,E2 29790.897} C_VEL
LIN {X 0,Y 639.901,Z 1294.786,A -85,B 0,C 180,E1 29789.195,E2 29789.195} C_VEL
